		//Success
		IF NOT FB_MBReadInputs_Read.bBusy AND NOT FB_MBReadInputs_Read.bError THEN
			bRead := FALSE;
			bError := FALSE;
		END_IF	
		
		bRead := WORD_TO_BOOL(wRead);
	
	3: //Read Holding reg
		
		FB_MBReadRegs_Read(
		sIPAddr:= sIPAddr, 
		nTCPPort:= nTCPPort, 
		nUnitID:= nUnitID, 
		nQuantity:= 1 + nAddQuantity, 
		nMBAddr:= mBusAdr, 
		cbLength:= SIZEOF(aWordArrayRead), 
		pDestAddr:= ADR(aWordArrayRead), 
		bExecute:= bRead, 
		tTimeout:= tTimeout, 
		bBusy=> , 
		bError=> , 
		nErrId=> , 
		cbRead=> );
	
		//Error 
		IF FB_MBReadRegs_Read.bError THEN
			bRead := FALSE;
			bError := TRUE;
		END_IF
		
		//Success
		IF NOT FB_MBReadRegs_Read.bBusy AND NOT FB_MBReadRegs_Read.bError THEN
			bRead := FALSE;
			bError := FALSE;
		END_IF	
				
		//Skriv värdet
		IF bRead32bit THEN 
			IF bSwap THEN
				rRead := fWordToReal(aWordArrayRead);
			ELSE
				aWordArrayNoSwap[0] := aWordArrayRead[1];
				aWordArrayNoSwap[1] := aWordArrayRead[0];
 				rRead := fWordToReal(aWordArrayNoSwap);
			END_IF
		ELSE
			rRead := fSignedConverter(aWordArrayRead[0]);
		END_IF;
		
	4: //Read input registers
		
		FB_MBReadInputRegs_Read(
		sIPAddr:= sIPAddr, 
		nTCPPort:= nTCPPort, 
		nUnitID:= nUnitID, 
		nQuantity:= 1 + nAddQuantity, 
		nMBAddr:= mBusAdr, 
		cbLength:= SIZEOF(aWordArrayRead), 
		pDestAddr:= ADR(aWordArrayRead), 
		bExecute:= bRead, 
		tTimeout:= tTimeout, 
		bBusy=> , 
		bError=> , 
		nErrId=> , 
		cbRead=> );
	
		//Error 
		IF FB_MBReadInputRegs_Read.bError THEN
			bRead := FALSE;
			bError := TRUE;
		END_IF
		
		//Success
		IF NOT FB_MBReadInputRegs_Read.bBusy AND NOT FB_MBReadInputRegs_Read.bError THEN
			bRead := FALSE;
			bError := FALSE;
		END_IF	
	
		//Skriv värdet
		IF bRead32bit THEN 
			IF bSwap THEN
				rRead := fWordToReal(aWordArrayRead);
			ELSE
				aWordArrayNoSwap[0] := aWordArrayRead[1];
				aWordArrayNoSwap[1] := aWordArrayRead[0];
 				rRead := fWordToReal(aWordArrayNoSwap);
			END_IF
		ELSE
			rRead := fSignedConverter(aWordArrayRead[0]);
		END_IF;

END_CASE

bBusy := FB_MBReadCoils_Read.bBusy OR FB_MBReadInputs_Read.bBusy OR FB_MBReadRegs_Read.bBusy OR FB_MBReadInputRegs_Read.bBusy;

END_FUNCTION_BLOCK

// oaksModbusLibrary/Datahantering/fWordToReal
//OAKS AB
//2020-03-18
//Funtionsblock för att lägga ihop två separata word till en real 
FUNCTION fWordToReal : REAL
VAR_INPUT

wAwords : ARRAY  [0..1] OF WORD;
END_VAR
VAR
	union1 : uRealToTwoWORD;
END_VAR

union1.wTest[0] := wAwords[0];
union1.wTest[1] := wAwords[1];

fWordToReal := union1.rTest;

END_FUNCTION

// oaksModbusLibrary/Datahantering/fbReadWriteCoilRegBool
//Oaks AB
//2022-08-22
//Funktionsblock för läsning av coil register (modbus funktion 15). Värde skrivs endast då skriv värde avviker från återläst värde. Används ej på EEPROM minnen, då det riskerar att skriva sönder dem. Använd istället block med återläsning av värden.
//Läsning och skrivning sker i sekvens.
//Två larmutgångar. En via puls kopplas till tex. en TOF för egen larmhantering. En via inställd larmtid. Skall summalarm i skåp tändas vid fel kopplas någon av utgångarna till externt fbAlarm. 

FUNCTION_BLOCK fbReadWriteCoilRegBool
VAR_INPUT
	sIPAddr : STRING := ''; //Ip-adress
	nTCPPort : UINT; //Port
	nUnitID : UINT; //Modbus-ID
	mBusAdr : UINT; //Holding adress att läsa/skriva
	bEnable : BOOL := TRUE; //Flanktriggad
	tTimeout : TIME := T#5S;
	bBool : BOOL := FALSE; //Värde att skriva
			
END_VAR
VAR_OUTPUT
	bError : BOOL; //Puls (Använd för egen larmhantering)
	bBusy : BOOL; //Upptagen
	bSuccess : BOOL := FALSE; //Lyckad cykel
END_VAR

VAR
	bEnableInternal : BOOL := TRUE;
	iStep : INT := 0;
	fbReadRegs_1: FB_MBReadCoils;
	fbWriteCoils_Write: FB_MBWriteCoils;
	bRead : BOOL; //Värde återläst
	bWrite : BOOL; //Värde att skriva
	R_TRIG_Start : R_TRIG; 

	FB_MBWriteSingleCoil_Write: INT;
	
END_VAR

//Flanktriggning
R_TRIG_Start(CLK:= bEnable, Q=> bEnableInternal);

//Läs och skriv värden
CASE iStep OF
	
	0: //Start
		bSuccess := FALSE;
		bBusy := FALSE;
		
		IF bEnableInternal THEN
			iStep := 1;
			bError := FALSE;
		END_IF
		
	1: //Läs data
		bBusy := TRUE;
		
		fbReadRegs_1(
				sIPAddr:= sIPAddr, 
				nTCPPort:= INT_TO_UINT(nTCPPort), 
				nUnitID:= INT_TO_BYTE(nUnitID), 
				nQuantity:= 1, 
				nMBAddr:= UINT_TO_WORD(mBusAdr), 
				cbLength:= SIZEOF(bRead), 
				pDestAddr:= ADR(bRead), 
				bExecute:= TRUE,
				tTimeout:= tTimeout, 
				bBusy=> , 
				bError=> , 
				nErrId=> , 
				cbRead=> );
				
		//Error 
		IF fbReadRegs_1.bError THEN
			fbReadRegs_1(bExecute := FALSE);
			iStep := 99;
		END_IF
	
		//Gå till nästa steg
		IF NOT fbReadRegs_1.bBusy AND NOT fbReadRegs_1.bError THEN
			fbReadRegs_1(bExecute := FALSE);
			bError := FALSE;
			iStep := 2;
		END_IF;

	2: //Skriv data
	
		bWrite := bBool;
	
			//15 Force Multiple Coils
			IF bWrite <> bRead THEN
				fbWriteCoils_Write.bExecute := TRUE;
			ELSE
				fbWriteCoils_Write.bExecute := FALSE;
			END_IF;
			
				fbWriteCoils_Write(
					sIPAddr:= sIPAddr, 
					nTCPPort:= INT_TO_UINT(nTCPPort), 
					nUnitID:= INT_TO_BYTE(nUnitID), 
					nQuantity:= 1, 
					nMBAddr:= UINT_TO_WORD(mBusAdr),
					cbLength:= SIZEOF(bWrite), 
					pSrcAddr:= ADR(bWrite), 
					bExecute:= , 
					tTimeout:= tTimeout, 
					bBusy=> , 
					bError=> , 
					nErrId=> );
			
			//Felhantering
			IF fbWriteCoils_Write.bError THEN
				fbWriteCoils_Write(bExecute := FALSE);
				iStep := 99;
			END_IF
			
			//Nästa steg
			IF NOT fbWriteCoils_Write.bBusy AND NOT fbWriteCoils_Write.bError THEN
				fbWriteCoils_Write(bExecute := FALSE);
				bError := FALSE;
				bSuccess := TRUE; //Lyckad cykel
				iStep := 0;
			END_IF;
				
		99: //Felhantering total
			bError := TRUE;
			iStep := 0;
END_CASE

END_FUNCTION_BLOCK

// oaksModbusLibrary/Datahantering/fbReadWriteHoldingRegReal
//Oaks AB
//2022-02-08
//Funktionsblock för läsning av holding register. Värde skrivs endast då skriv värde avviker från återläst värde. Används ej på EEPROM minnen, då det riskerar att skriva sönder dem. Använd istället block med återläsning av värden.
//Real med skalning direkt anges på block, med inbyggd hantering av negativa värden. Läsning och skrivning sker i sekvens.
//Två larmutgångar. En via puls kopplas till tex. en TOF för egen larmhantering. En via inställd larmtid. Skall summalarm i skåp tändas vid fel kopplas någon av utgångarna till externt fbAlarm. 

FUNCTION_BLOCK fbReadWriteHoldingRegReal
VAR_INPUT
	sIPAddr : STRING := ''; //Ip-adress
	nTCPPort : UINT; //Port
	nUnitID : UINT; //Modbus-ID
	mBusAdr : UINT; //Holding adress att läsa/skriva
	bEnable : BOOL := TRUE; //Flanktriggad
	tTimeout : TIME := T#5S;
	rReal : REAL := 0; //Värde att skriva
	uiFaktor : REAL := 1; //Skalning
	
END_VAR
VAR_OUTPUT
	bError : BOOL; //Puls (Använd för egen larmhantering)
	bBusy : BOOL; //Upptagen
	bSuccess : BOOL := FALSE; //Lyckad cykel
END_VAR

VAR
	bEnableInternal : BOOL := TRUE;
	iStep : INT := 0;
	fbReadRegs_1: FB_MBReadRegs;
	fbWriteSingleReg_1: FB_MBWriteSingleReg;
	wRead : WORD; //Värde återläst
	wWrite : WORD; //Värde att skriva
	R_TRIG_Start : R_TRIG; 
END_VAR

//Flanktriggning
R_TRIG_Start(CLK:= bEnable, Q=> bEnableInternal);

//Läs och skriv värden
CASE iStep OF
	
	0: //Start
		bSuccess := FALSE;
		bBusy := FALSE;
		
		IF bEnableInternal THEN
			iStep := 1;
			bError := FALSE;
		END_IF
		
	1: //Läs data
		bBusy := TRUE;
		
		fbReadRegs_1(
				sIPAddr:= sIPAddr, 
				nTCPPort:= INT_TO_UINT(nTCPPort), 
				nUnitID:= INT_TO_BYTE(nUnitID), 
				nQuantity:= 1, 
				nMBAddr:= UINT_TO_WORD(mBusAdr), 
				cbLength:= SIZEOF(wRead), 
				pDestAddr:= ADR(wRead), 
				bExecute:= TRUE,
				tTimeout:= tTimeout, 
				bBusy=> , 
				bError=> , 
				nErrId=> , 
				cbRead=> );
	
		//Error 
		IF fbReadRegs_1.bError THEN
			fbReadRegs_1(bExecute := FALSE);
			iStep := 99;
		END_IF
	
		//Gå till nästa steg
		IF NOT fbReadRegs_1.bBusy AND NOT fbReadRegs_1.bError THEN
			fbReadRegs_1(bExecute := FALSE);
			bError := FALSE;
			iStep := 2;
		END_IF;

	2: //Skriv data
		//Konvertera REAL till WORD. 
		wWrite := fRealToWord(rReal, uiFaktor);
		//Skriv om värden skiljer sig
		IF wWrite <> wRead THEN
			fbWriteSingleReg_1(
				sIPAddr:= sIPAddr, 
				nTCPPort:= INT_TO_UINT(nTCPPort), 
				nUnitID:= INT_TO_BYTE(nUnitID), 
				nMBAddr:= UINT_TO_WORD(mBusAdr),
				nValue:= wWrite, 
				bExecute:= TRUE, 
				tTimeout:= tTimeout , 
				bBusy=> , 
				bError=> , 
				nErrId=> );
		//Annars börja om
		ELSE 
			iStep := 0;
		END_IF;
		
		//Felhantering
		IF fbWriteSingleReg_1.bError THEN
			fbWriteSingleReg_1(bExecute := FALSE);
			iStep := 99;
		END_IF
		
		//Nästa steg
		IF NOT fbWriteSingleReg_1.bBusy AND NOT fbWriteSingleReg_1.bError THEN
			fbWriteSingleReg_1(bExecute := FALSE);
			bError := FALSE;
			bSuccess := TRUE; //Lyckad cykel
			iStep := 0;
		END_IF;
			
		99: //Felhantering total
			bError := TRUE;
			iStep := 0;
END_CASE

END_FUNCTION_BLOCK

// oaksModbusLibrary/EBM Papst/fbEbmPapst
//OAKS AB
//2023-06-28
//Ver. 1.0
//Modbusblock för ebmpapst fläkt.
FUNCTION_BLOCK fbEbmPapst
VAR_INPUT
	sIPAddr : STRING := ''; 
	nTCPPort : UINT;
	nUnitID : UINT :=1;
	iModbusLoop : INT :=1; //Modbusslinga
			
END_VAR
VAR_OUTPUT
	RPM AT %M* : REAL;//Varvtal~wp:[unit]RPM[format]0[trendoptions]i:300
	U1 AT %M* : REAL;//Spänning~wp:[unit]V[format]0[trendoptions]i:300
	I1 AT %M* : REAL;//Ampere~wp:[unit]A[format]0.0[trendoptions]i:300	
	P1 AT %M* : REAL;//Effekt~wp:[unit]kW[format]0.0[trendoptions]i:300		
	PV8 AT %M* : STRING;//Modbus konfiguering~wp:
	FAULT AT %M* : BOOL;//Kommunikationsfel~wp:[alarmoptions]p:2
	
END_VAR
VAR
	offset : UINT;
	rTemp1 : REAL;
	rTemp2 : REAL;
	bSekvensFlagga : BOOL;
			
	FB_MBReadRegs_ArrReadRegs1 : FB_MBReadRegs;
	FB_MBReadRegs_ArrReadRegs2 : FB_MBReadRegs;
	FB_MBReadRegs_ArrReadInputsRegs1 : FB_MBReadInputRegs;
	FB_MBReadRegs_ArrReadInputsRegs2 : FB_MBReadInputRegs;

	wArrReadRegs1 : ARRAY [0..0] OF WORD; //ReadRegs
	wArrReadRegs2 : ARRAY [0..1] OF WORD; //ReadRegs
	wArrReadInputsRegs1 : ARRAY [0..9] OF WORD; //ReadInputsRegs
	wArrReadInputsRegs2 : ARRAY [0..9] OF WORD; //ReadInputsRegs
		
	//Kommunikationsfel
	fbKommTof : tof; 
	fbKommTon : fbAlarm;
	
	sIP: STRING(255);
	sPort: STRING(255);
	sModbusID: STRING(255);
	sModbusLoop: STRING(255);
	sTemp : STRING(255);
	
END_VAR

//General
	offset := 0;
//Sekvens	
	bSekvensFlagga := oaksGVL.aBModbusSekvens[iModbusLoop] = UINT_TO_INT(nUnitID);
//Modbus konfiguering
	sIP := CONCAT (SIPAddr, '');
	sPort := CONCAT ('<br>Port: ', UINT_TO_STRING(nTCPPort)); 								
	sModbusID := CONCAT('<br>ID: ', UINT_TO_STRING(nUnitID));
	sModbusLoop := CONCAT('<br>Loop: ', INT_TO_STRING(iModbusLoop));	

	sTemp := sIP;
	sTemp := CONCAT(sTemp, sPort);
	sTemp := CONCAT(sTemp, sModbusID);
	sTemp := CONCAT(sTemp, sModbusLoop);
	
	PV8 := sTemp;

///////////////		
//READ
///////////////		
	
	//Read Register D119
	FB_MBReadRegs_ArrReadRegs1(
	sIPAddr:= sIpAddr, 
	nTCPPort:= (nTCPPort),
	nUnitID:= UINT_TO_BYTE(nUnitID),  
	nQuantity:= 1, 
	nMBAddr:= 53529 + offset, 
	cbLength:= SIZEOF(wArrReadRegs1),  
	pDestAddr:= ADR(wArrReadRegs1), 
	bExecute:= bSekvensFlagga, 
	tTimeout:= T#10S, 
	bBusy=> , 
	bError=> , 
	nErrId=> , 
	cbRead=> );

	//Read Register D1A0-D1A1
	FB_MBReadRegs_ArrReadRegs2(
	sIPAddr:= sIpAddr, 
	nTCPPort:= (nTCPPort),
	nUnitID:= UINT_TO_BYTE(nUnitID),  
	nQuantity:= 2, 
	nMBAddr:= 53664 + offset, 
	cbLength:= SIZEOF(wArrReadRegs2),  
	pDestAddr:= ADR(wArrReadRegs2), 
	bExecute:= bSekvensFlagga, 
	tTimeout:= T#10S, 
	bBusy=> , 
	bError=> , 
	nErrId=> , 
	cbRead=> );	

	//Read Inputs D010-D019
	FB_MBReadRegs_ArrReadInputsRegs1(
	sIPAddr:= sIpAddr, 
	nTCPPort:= (nTCPPort), 
	nUnitID:= UINT_TO_BYTE(nUnitID), 
	nQuantity:= 9, 
	nMBAddr:= 53264 + offset,
	cbLength:= SIZEOF(wArrReadInputsRegs1), 
	pDestAddr:= ADR(wArrReadInputsRegs1), 
	bExecute:= bSekvensFlagga,
	tTimeout:= T#10S, 
	bBusy=> , 
	bError=> , 
	nErrId=> , 
	cbRead=> );	
	
	//Read Inputs D01A-D023
	FB_MBReadRegs_ArrReadInputsRegs2(
	sIPAddr:= sIpAddr, 
	nTCPPort:= (nTCPPort), 
	nUnitID:= UINT_TO_BYTE(nUnitID), 
	nQuantity:= 9, 
	nMBAddr:= 53274 + offset,
	cbLength:= SIZEOF(wArrReadInputsRegs2), 
	pDestAddr:= ADR(wArrReadInputsRegs2), 
	bExecute:= bSekvensFlagga,
	tTimeout:= T#10S, 
	bBusy=> , 
	bError=> , 
	nErrId=> , 
	cbRead=> );		

		//Values
		RPM := ((wArrReadInputsRegs1[0]*wArrReadRegs1[0])/64000); //D010 - Actual speed, Res.:1, Unit:rpm
		//wArrReadInputsRegs1[1]; //D011 - Notor status, Res.:-, Unit:-
		//wArrReadInputsRegs1[2]; //D012 - Warning, Res.:-, Unit:-
		U1 := (((wArrReadInputsRegs1[3]*(wArrReadRegs2[0]*20))/256)*0.001); //D013 - DC-link voltage, Res.:1, Unit:V
		I1 := (((wArrReadInputsRegs1[4]*(wArrReadRegs2[1]*2))/256)*0.001); //D014 - DC-link current, Res.:0.1, Unit:A
		//wArrReadInputsRegs1[5]; //D015 - Modul temperature, Res.:0.1, Unit:ºC
		//wArrReadInputsRegs1[6]; //D016 - Motor temperature, Res.:0.1, Unit:ºC
		//wArrReadInputsRegs1[7]; //D017 - Electronics temperature, Res.:0.1, Unit:ºC
		//wArrReadInputsRegs1[8]; //D018 - Current direction of rotation, Res.:-, Unit:-
		//wArrReadInputsRegs1[9]; //D019 - Current modulation level, Res.:-, Unit:-
	
		//wArrReadInputsRegs2[0]; //D01A - Current set value, Res.:-, Unit:-
		//wArrReadInputsRegs2[1]; //D01B - Actual sensor value, Res.:-, Unit:-
		//wArrReadInputsRegs2[2]; //D01C - Enable input status, Res.:-, Unit:-
		//wArrReadInputsRegs2[3]; //D01D - Current parameter set, Res.:-, Unit:-
		//wArrReadInputsRegs2[4]; //D01E - Current contol function, Res.:-, Unit:-
		//wArrReadInputsRegs2[5]; //D01F - Reserved, Res.:-, Unit:-
		//wArrReadInputsRegs2[6]; //D020 - Reserved, Res.:-, Unit:-
		rTemp1 := ((wArrReadRegs2[0]*20)*0.001);
		rTemp2 := ((wArrReadRegs2[1]*2)*0.001);
		P1 := ((((wArrReadInputsRegs2[7]*rTemp1)*rTemp2)/65536)*0.001); //D021 - Current power, Res.:0.1, Unit:kW 
		//wArrReadInputsRegs2[8]; //D022 - Reserved, Res.:-, Unit:-
		//wArrReadInputsRegs2[9]; //D023 - Acyual sensor value 1, Res.:-, Unit:-
	
//Communication error
	fbKommTof(IN:=FB_MBReadRegs_ArrReadInputsRegs1.bError , PT:=T#60S , Q=> , ET=> );
	fbKommTon(bInput:=fbKommTof.Q , tAlarmDelay:=T#20M , bAutoReset:= , bAlarmOutput=> );
	FAULT :=fbKommTon.bAlarmOutput;
		
//Write busy	
	oaksgvl.aBModbusBusyFlagga[iModbusLoop,nUnitID] := FB_MBReadRegs_ArrReadInputsRegs1.bBusy;

END_FUNCTION_BLOCK

// oaksModbusLibrary/EcoGuard/fbEcocomTemperature
//OAKS AB
//2020-03-18
// Funktionsblock för kommunikation  rumstemperatur från Ecoguard Ecocom
FUNCTION_BLOCK fbEcocomTemperature
VAR_INPUT
	sIpNUmber									: STRING(32);						// Ip nummer för Slav
	nTcpPort									: UINT := 502;					// Modbus port
	nUnitID 									: BYTE := 1;
	nAdressMaxTemperature						: UINT; 
	nAdressAvgTemperature						: UINT; 
	nAdressMinTemperature						: UINT; 
	tCommAlarmDelay : TIME := T#30M; // Tid för kommunikationsfelslarm.
	tToggleTime 	: TIME := T#60S; // ange hur ofta frågor skall ställas till Elvacon.
	tTimeout 		: TIME := T#58S; // inställd timeout-tid.
END_VAR
VAR_OUTPUT
	PV AT %M* : REAL;//Medel rumstemperatur hämtat från Ecoguard Ecocom~wp:[unit]°C[format]0.0[trendoptions]i:300
	PV1 AT %M* : REAL;//Högsta rumstemperatur hämtat från Ecoguard Ecocom~wp:[unit]°C[format]0.0[trendoptions]i:300
	PV2 AT %M* : REAL;//Lägsta rumstemperatur hämtat från Ecoguard Ecocom~wp:[unit]°C[format]0.0[trendoptions]i:300
	FAULT AT %M* : BOOL;//Kommunikationsfel~wp:
	PV8 AT %M* : STRING;//Modbus konfiguering~wp:
END_VAR
VAR
	rTemp : REAL;	

	sIP: STRING(255);
	sPort: STRING(255);
	sModbusID: STRING(255);
	sMaxtemp: STRING(255);
	sMedeltemp: STRING(255);
	sMintemp: STRING(255);
	sTemp : STRING(255);	

	fbKommTof : TOF;	
	fbKommTon : TON;
	FB_MBReadRegsAvg : FB_MBReadRegs;
	FB_MBReadRegsMax : FB_MBReadRegs;
	FB_MBReadRegsMin : FB_MBReadRegs;
	
	wInternalTempAvg : 	WORD; 
	wInternalTempMax : 	WORD; 
	wInternalTempMin : 	WORD; 
	fbToggle01: fbToggle;
	
END_VAR

//Modbus konfiguering
	sIP := CONCAT (sIpNUmber, '');
	sPort := CONCAT ('<br>Port: ', UINT_TO_STRING(nTCPPort)); 	
	sMaxtemp := CONCAT('<br>Adress maxtemperatur: ', INT_TO_STRING(nAdressMaxTemperature));						
	sMedeltemp := CONCAT('<br>Adress medeltemperatur: ', INT_TO_STRING(nAdressAvgTemperature));	
	sMintemp := CONCAT('<br>Adress mintemperatur: ', INT_TO_STRING(nAdressMinTemperature));
	
	sTemp := sIP;
	sTemp := CONCAT(sTemp, sPort);
	sTemp := CONCAT(sTemp, sMaxtemp);
	sTemp := CONCAT(sTemp, sMedeltemp);
	sTemp := CONCAT(sTemp, sMintemp);
	
	PV8 := sTemp;

	fbToggle01(bStart:=TRUE , tTimeOn:=tToggleTime , tTimeOff:=tToggleTime , bOutput=> );

	fbKommTof(IN:=FB_MBReadRegsAvg.bError OR FB_MBReadRegsMin.bError OR FB_MBReadRegsMax.bError , PT:=T#20S , Q=> , ET=> );
	fbKommTon(IN:=fbKommTof.Q , PT:=tCommAlarmDelay , Q=>FAULT , ET=> );
	// Hämta medel temperatur
	FB_MBReadRegsAvg(
	sIPAddr:= sIpNUmber, 
	nTCPPort:=nTcpPort , 
	nUnitID:=nUnitID , 
	nQuantity:=1 , 
	nMBAddr:= nAdressAvgTemperature, 
	cbLength:=SIZEOF(wInternalTempAvg) , 
	pDestAddr:=ADR(wInternalTempAvg) , 
	bExecute:=fbToggle01.bOutput , 
	tTimeout:=tTimeout , 
	bBusy=> , 
	bError=> , 
	nErrId=> , 
	cbRead=> );
	
	rTemp := fSignedConverter(wInternalTempAvg); 
	
	PV := rTemp / 10;
	// Hämta max temperatur
	FB_MBReadRegsMax(
	sIPAddr:= sIpNUmber, 
	nTCPPort:=nTcpPort , 
	nUnitID:=nUnitID , 
	nQuantity:=1 , 
	nMBAddr:= nAdressMaxTemperature, 
	cbLength:=SIZEOF(wInternalTempMax) , 
	pDestAddr:=ADR(wInternalTempMax) , 
	bExecute:=fbToggle01.bOutput , 
	tTimeout:=tTimeout , 
	bBusy=> , 
	bError=> , 
	nErrId=> , 
	cbRead=> );
	
	rTemp := fSignedConverter(wInternalTempMax); 
	
	PV1 := rTemp / 10;
	
	// Hämta min temperatur
	FB_MBReadRegsMin(
	sIPAddr:= sIpNUmber, 
	nTCPPort:=nTcpPort , 
	nUnitID:=nUnitID , 
	nQuantity:=1 , 
	nMBAddr:= nAdressMinTemperature, 
	cbLength:=SIZEOF(wInternalTempMin) , 
	pDestAddr:=ADR(wInternalTempMin) , 
	bExecute:=fbToggle01.bOutput , 
	tTimeout:=tTimeout , 
	bBusy=> , 
	bError=> , 
	nErrId=> , 
	cbRead=> );
	
	rTemp := fSignedConverter(wInternalTempMin); 
	
	PV2 := rTemp / 10;

END_FUNCTION_BLOCK

// oaksModbusLibrary/Elvaco/CME3100/Givare/fbElvacoTemperature
//OAKS AB
//2020-03-18
// Funktionsblock för kommunikation  via four-byte swapped float rumstemperatur från Elvaco CME3100
FUNCTION_BLOCK fbElvacoTemperature
VAR_INPUT
	sIpNUmber								: 		STRING(32);						// Ip nummer för Slav
	nTcpPort								: 		UINT := 502;					// Modbus port
	iModbusLoop : REFERENCE TO INT := 0; // Vill man att läsningarna ska ske givare för givare skapa en INT-variabel med värdet 16 som du sedan knyter hit. Läsningarna kommer då att ske efter modbussekvens 16. Knyter man inget här läses värdena efter inställd tid i tToggleTime samtidigt vilket kan bli problematiskt vid väldigt många samtidiga läsningar.
	nAdressTemperature						: UINT; 
	tCommAlarmDelay : TIME := T#30M; // Tid för kommunikationsfelslarm.
	tToggleTime : TIME := T#60S; // ange hur ofta frågor skall ställas till Elvacon. Denna används inte om något är knutet till iModbusLoop.
	tTimeout : TIME := T#58S; // inställd timeout-tid. Knyter man något på iModbusLoop är timeout-tiden 5 sekunder innan den går vidare.
	iSecId : DINT := 0;//Sekundär-ID
END_VAR
VAR_OUTPUT
	PV AT %M* : REAL;//Rumstemperatur~wp:[unit]°C[format]0.0[trendoptions]i:300
	FAULT AT %M* : BOOL;//Kommunikationsfel~wp:
	PV8 AT %M* : STRING;//Modbus konfiguering~wp:
END_VAR
VAR
	fbDifferenceCheckTemp: fbDifferenceCheck;
	fbAlarmTemp : fbAlarm;
	fbTonDifferenceCheck : TON;

	tTimeoutIntern : TIME;
	bStartaLasningTemperatur	: BOOL;

	bSekvensFlagga : BOOL;	

	sIP: STRING(255);
	sPort: STRING(255);
	sModbusID: STRING(255);
	sModbusLoop: STRING(255);
	sSecId : STRING(255);
	sTemp : STRING(255);

	fbKommTof : TOF;	
	fbKommTon : TON;
	FB_MBReadRegs01 : FB_MBReadRegs;
	wInternalTemp : ARRAY[0..1] OF	WORD; 
	fbToggle01: fbToggle;
	
	uRealToTwoWORD01 : uRealToTwoWORD;
END_VAR
VAR PERSISTENT
	tAlarmDelayDifferenceCheck : TIME := T#48H;
END_VAR

VAR_INPUT PERSISTENT
	AREAT AT %M* : INT; //Yta rumstemperatur~wp:
END_VAR


	IF __ISVALIDREF(iModbusLoop) THEN 
		IF iModbusLoop < 16 OR iModbusLoop > 16 THEN
			iModbusLoop := 16;
		END_IF;
		bSekvensFlagga := oaksGVL.aBModbusSekvens[iModbusLoop] = UINT_TO_INT(nAdressTemperature);
		fbToggle01(bStart:=FALSE , tTimeOn:=tToggleTime , tTimeOff:=tToggleTime , bOutput=> );
		tTimeoutIntern := T#5S;
	ELSE
		fbToggle01(bStart:=TRUE , tTimeOn:=tToggleTime , tTimeOff:=tToggleTime , bOutput=> );
		tTimeoutIntern := tTimeout;
	END_IF;
	bStartaLasningTemperatur := bSekvensFlagga OR fbToggle01.bOutput;

//Modbus konfiguering
	sIP := CONCAT (sIpNUmber, '');
	sPort := CONCAT ('<br>Port: ', UINT_TO_STRING(nTCPPort)); 						
	sModbusLoop := CONCAT('<br>Adress: ', INT_TO_STRING(nAdressTemperature));
	sSecId := CONCAT('<br>Sekundär-Id: ', DINT_TO_STRING(iSecId));

	sTemp := sIP;
	sTemp := CONCAT(sTemp, sPort);
	sTemp := CONCAT(sTemp, sModbusLoop);
	
	//Sekundär-Id
	IF iSecID > 0 THEN
		sTemp := CONCAT(Stemp,sSecId);
	ELSE 
		sTemp := STemp;
	END_IF
		
	PV8 := sTemp;

	fbKommTof(IN:=FB_MBReadRegs01.bError , PT:=T#20S , Q=> , ET=> );
	fbKommTon(IN:=fbKommTof.Q , PT:=tCommAlarmDelay , Q=>FAULT , ET=> );
	
	fbDifferenceCheckTemp(rPv:=PV );
	fbTonDifferenceCheck(IN:=NOT fbDifferenceCheckTemp.bDifference , PT:=tAlarmDelayDifferenceCheck , Q=> , ET=> );
	fbAlarmTemp(bInput:= fbTonDifferenceCheck.Q OR fbKommTon.Q , tAlarmDelay:=T#0S , bAutoReset:=TRUE , bAlarmOutput=>FAULT);

	FB_MBReadRegs01(
	sIPAddr:= sIpNUmber, 
	nTCPPort:=nTcpPort , 
	nUnitID:=1 , 
	nQuantity:=2 , 
	nMBAddr:= nAdressTemperature, 
	cbLength:=SIZEOF(wInternalTemp) , 
	pDestAddr:=ADR(wInternalTemp) , 
	bExecute:=bStartaLasningTemperatur , 
	tTimeout:=tTimeoutIntern , 
	bBusy=> , 
	bError=> , 
	nErrId=> , 
	cbRead=> );
	
	uRealToTwoWORD01.wTest[0] :=wInternalTemp [0];
	uRealToTwoWORD01.wTest[1] :=wInternalTemp [1];
	PV := uRealToTwoWORD01.rTest;
	
IF __ISVALIDREF(iModbusLoop) THEN 
	//Write busy
	oaksgvl.aBModbusBusyFlaggaAdresser[iModbusLoop-15,nAdressTemperature] := FB_MBReadRegs01.bBusy;
END_IF

END_FUNCTION_BLOCK

// oaksModbusLibrary/Elvaco/CME3100/Givare/fbElvacoTemperatureCo2
FUNCTION_BLOCK fbElvacoTemperatureCo2 EXTENDS fbElvacoTemperature
VAR_INPUT
	nAdressCo2		: UINT; 
END_VAR
VAR_OUTPUT
	PV1 AT %M* : REAL;//Koldioxidhalt~wp:[unit]ppm[format]0[trendoptions]i:300
END_VAR
VAR
	FB_MBReadRegs02 : FB_MBReadRegs;
	
	wInternalCo2	 : ARRAY[0..1] OF	WORD; 
	uRealToTwoWORD02 : uRealToTwoWORD;
END_VAR

VAR_INPUT PERSISTENT
	AREACO2 AT %M* : INT; //Yta koldioxid~wp:
END_VAR

	SUPER^();

	FB_MBReadRegs02(
	sIPAddr:= sIpNUmber, 
	nTCPPort:=nTcpPort , 
	nUnitID:=1 , 
	nQuantity:=2 , 
	nMBAddr:= nAdressCo2, 
	cbLength:=SIZEOF(wInternalCo2) , 
	pDestAddr:=ADR(wInternalCo2) , 
	bExecute:=bStartaLasningTemperatur , 
	tTimeout:=tTimeoutIntern , 
	bBusy=> , 
	bError=> , 
	nErrId=> , 
	cbRead=> );
	
	uRealToTwoWORD02.wTest[0] :=wInternalCo2 [0];
	uRealToTwoWORD02.wTest[1] :=wInternalCo2 [1];
	PV1 := uRealToTwoWORD02.rTest;

END_FUNCTION_BLOCK

// oaksModbusLibrary/Elvaco/CME3100/Givare/fbElvacoTemperatureHumidity
FUNCTION_BLOCK fbElvacoTemperatureHumidity EXTENDS fbElvacoTemperature
VAR_INPUT
	nAdressHumidity		: UINT; 
END_VAR
VAR_OUTPUT
	PV1 AT %M* : REAL;//Fukthalt~wp:[unit]rH%[trendoptions]i:300
END_VAR
VAR
	FB_MBReadRegs02 : FB_MBReadRegs;
	
	wInternalHumidity	 : ARRAY[0..1] OF	WORD; 
	uRealToTwoWORD02 : uRealToTwoWORD;
END_VAR

VAR_INPUT PERSISTENT
	AREAH AT %M* : INT; //Yta fuktighet~wp:
END_VAR

	SUPER^();

	FB_MBReadRegs02(
	sIPAddr:= sIpNUmber, 
	nTCPPort:=nTcpPort , 
	nUnitID:=1 , 
	nQuantity:=2 , 
	nMBAddr:= nAdressHumidity, 
	cbLength:=SIZEOF(wInternalHumidity) , 
	pDestAddr:=ADR(wInternalHumidity) , 
	bExecute:=bStartaLasningTemperatur , 
	tTimeout:=tTimeoutIntern , 
	bBusy=> , 
	bError=> , 
	nErrId=> , 
	cbRead=> );
	
	uRealToTwoWORD02.wTest[0] :=wInternalHumidity [0];
	uRealToTwoWORD02.wTest[1] :=wInternalHumidity [1];
	PV1 := uRealToTwoWORD02.rTest;

END_FUNCTION_BLOCK

// oaksModbusLibrary/Elvaco/CME3100/Mätare/fbElvacoElectricMeter
//OAKS AB
//2020-05-12
//Funktionsblock för att läsa elmätare från Elvaco
FUNCTION_BLOCK fbElvacoElectricMeter
VAR_INPUT
	sIPAddr : STRING := ''; 
	nTCPPort : UINT;
	nAdressEnergy	: UINT;
	nAdressPower	: UINT; 
	tCommAlarmDelay : TIME := T#30M; // Tid för kommunikationsfelslarm.
	tToggleTime : TIME := T#10S; // ange hur ofta frågor skall ställas till Elvacon.
	tTimeout : TIME := T#8S; // inställd timeout-tid.
	iSecId : DINT := 0;//Sekundär-ID
	rScalePower : REAL :=1; //Skalning effekt
 	bActivateDifferenceCheck : BOOL := TRUE; // När denna är true utgår kommunikationsfelslarm ifall värdet ej ändrats på T#49D17H2M47S295MS (inställbart)
END_VAR
VAR_OUTPUT
	PV8 AT %M* : STRING;//Modbus konfiguering~wp:
	FAULT AT %M* : BOOL;//Kommunikationsfel~wp:
	PV AT %M* : REAL;//Energi~wp:[unit]kWh[format]0.0[trendoptions]i:300
	PV1 AT %M* : REAL;//Effekt~wp:[unit]kW[format]0.0[trendoptions]i:300
		
END_VAR
VAR
	fbDifferenceCheckValue: fbDifferenceCheck;
	fbAlarmValue : fbAlarm;	
	fbTonDifferenceCheck : TON;

	offset : WORD;
	rTemp : REAL;
	//iTemp : UINT;
	fbToggle01: fbToggle;	
	
	FB_MBReadRegs_Energy : FB_MBReadRegs;
	FB_MBReadRegs_Power : FB_MBReadRegs;
	
	rPowerRead : REAL;	
	
	//Kommunikationsfel
	fbKommTof : tof; 
	fbKommTon : fbAlarm;
	
	sIP: STRING(255);
	sPort: STRING(255);
	sModbusID: STRING(255);
	sModbusLoop: STRING(255);
	sTemp : STRING(255);
	sSecId : STRING(255);
END_VAR
VAR PERSISTENT
	tAlarmDelayDifferenceCheck : TIME := T#49D17H2M47S295MS;
END_VAR

//Modbus konfiguering
	sIP := CONCAT (sIPAddr, '');
	sPort := CONCAT ('<br>Port: ', UINT_TO_STRING(nTCPPort));
	sSecId := CONCAT('<br>Sekundär-Id: ', DINT_TO_STRING(iSecId));

	sTemp := sIP;
	sTemp := CONCAT(sTemp, sPort);
	sTemp := CONCAT(sTemp, sModbusLoop);
	
	//Sekundär-Id
	IF iSecID > 0 THEN
		sTemp := CONCAT(Stemp,sSecId);
	ELSE 
		sTemp := STemp;
	END_IF
		
	PV8 := sTemp;

///////////////		
//READ
///////////////		
	fbToggle01(bStart:=TRUE , tTimeOn:=tToggleTime , tTimeOff:=tToggleTime , bOutput=> );
	
	FB_MBReadRegs_Energy(
	sIPAddr:= sIpAddr, 
	nTCPPort:= INT_TO_UINT(nTCPPort), 
	nUnitID:= 1, 
	nQuantity:= 2, 
	nMBAddr:= nAdressEnergy + offset, 
	cbLength:= SIZEOF(PV), 
	pDestAddr:= ADR(PV), 
	bExecute:= fbToggle01.bOutput, 
	tTimeout:= tTimeout, 
	bBusy=> , 
	bError=> , 
	nErrId=> , 
	cbRead=> );
	
	FB_MBReadRegs_Power(
	sIPAddr:= sIpAddr, 
	nTCPPort:= INT_TO_UINT(nTCPPort), 
	nUnitID:= 1, 
	nQuantity:= 2, 
	nMBAddr:= nAdressPower + offset, 
	cbLength:= SIZEOF(rPowerRead), 
	pDestAddr:= ADR(rPowerRead), 
	bExecute:= fbToggle01.bOutput, 
	tTimeout:= tTimeout, 
	bBusy=> , 
	bError=> , 
	nErrId=> , 
	cbRead=> );
	
	//Skalning effekt då denna ofta kommer i W. 
	PV1 := rPowerRead * rScalePower;
	
//Communication error
	fbKommTof(IN:=FB_MBReadRegs_Energy.bError OR FB_MBReadRegs_Power.bError, PT:=T#20S , Q=> , ET=> );
	fbKommTon(bInput:=fbKommTof.Q , tAlarmDelay:=tCommAlarmDelay , bAutoReset:= , bAlarmOutput=> );
	fbDifferenceCheckValue(rPv:=PV );
	fbTonDifferenceCheck(IN:=NOT fbDifferenceCheckValue.bDifference , PT:=tAlarmDelayDifferenceCheck , Q=> , ET=> );
	fbAlarmValue(bInput:= (fbTonDifferenceCheck.Q AND bActivateDifferenceCheck) OR fbKommTon.bAlarmOutput, tAlarmDelay:=T#0S , bAutoReset:=TRUE , bAlarmOutput=>FAULT);

END_FUNCTION_BLOCK

// oaksModbusLibrary/Elvaco/CME3100/Mätare/fbElvacoElectricMeterEnergy
//OAKS AB
//2020-05-12
//Funktionsblock för att läsa elmätare från Elvaco
FUNCTION_BLOCK fbElvacoElectricMeterEnergy
VAR_INPUT
	sIPAddr : STRING := ''; 
	nTCPPort : UINT;
	nAdressEnergy	: UINT;
	tCommAlarmDelay : TIME := T#30M; // Tid för kommunikationsfelslarm.
	tToggleTime : TIME := T#10S; // ange hur ofta frågor skall ställas till Elvacon.
	tTimeout : TIME := T#8S; // inställd timeout-tid.
	iSecId : DINT := 0;//Sekundär-ID
	rScalePower : REAL :=1; //Skalning effekt
 	bActivateDifferenceCheck : BOOL := TRUE; // När denna är true utgår kommunikationsfelslarm ifall värdet ej ändrats på T#49D17H2M47S295MS (inställbart)
END_VAR
VAR_OUTPUT
	PV8 AT %M* : STRING;//Modbus konfiguering~wp:
	FAULT AT %M* : BOOL;//Kommunikationsfel~wp:
	PV AT %M* : REAL;//Energi~wp:[unit]kWh[format]0.0[trendoptions]i:300
			
END_VAR
VAR
	fbDifferenceCheckValue: fbDifferenceCheck;
	fbAlarmValue : fbAlarm;		
	fbTonDifferenceCheck : TON;
	offset : WORD;
	rTemp : REAL;
	//iTemp : UINT;
	fbToggle01: fbToggle;	
	
	FB_MBReadRegs_Energy : FB_MBReadRegs;
	
	//Kommunikationsfel
	fbKommTof : tof; 
	fbKommTon : fbAlarm;
	
	sIP: STRING(255);
	sPort: STRING(255);
	sModbusID: STRING(255);
	sModbusLoop: STRING(255);
	sTemp : STRING(255);
	sSecId : STRING(255);
END_VAR
VAR PERSISTENT
	tAlarmDelayDifferenceCheck : TIME := T#49D17H2M47S295MS;
END_VAR

//Modbus konfiguering
	sIP := CONCAT (sIPAddr, '');
	sPort := CONCAT ('<br>Port: ', UINT_TO_STRING(nTCPPort));
	sSecId := CONCAT('<br>Sekundär-Id: ', DINT_TO_STRING(iSecId));

	sTemp := sIP;
	sTemp := CONCAT(sTemp, sPort);
	sTemp := CONCAT(sTemp, sModbusLoop);
	
	//Sekundär-Id
	IF iSecID > 0 THEN
		sTemp := CONCAT(Stemp,sSecId);
	ELSE 
		sTemp := STemp;
	END_IF
		
	PV8 := sTemp;

///////////////		
//READ
///////////////		
	fbToggle01(bStart:=TRUE , tTimeOn:=tToggleTime , tTimeOff:=tToggleTime , bOutput=> );
	
	FB_MBReadRegs_Energy(
	sIPAddr:= sIpAddr, 
	nTCPPort:= INT_TO_UINT(nTCPPort), 
	nUnitID:= 1, 
	nQuantity:= 2, 
	nMBAddr:= nAdressEnergy + offset, 
	cbLength:= SIZEOF(PV), 
	pDestAddr:= ADR(PV), 
	bExecute:= fbToggle01.bOutput, 
	tTimeout:= tTimeout, 
	bBusy=> , 
	bError=> , 
	nErrId=> , 
	cbRead=> );
	
//Communication error
	fbKommTof(IN:=FB_MBReadRegs_Energy.bError, PT:=T#20S , Q=> , ET=> );
	fbKommTon(bInput:=fbKommTof.Q , tAlarmDelay:=tCommAlarmDelay , bAutoReset:= , bAlarmOutput=> );
	fbDifferenceCheckValue(rPv:=PV );
	fbTonDifferenceCheck(IN:=NOT fbDifferenceCheckValue.bDifference , PT:=tAlarmDelayDifferenceCheck , Q=> , ET=> );
	fbAlarmValue(bInput:= (fbTonDifferenceCheck.Q AND bActivateDifferenceCheck) OR fbKommTon.bAlarmOutput, tAlarmDelay:=T#0S , bAutoReset:=TRUE , bAlarmOutput=>FAULT);

END_FUNCTION_BLOCK

// oaksModbusLibrary/Elvaco/CME3100/Mätare/fbElvacoEnergyMeter
//OAKS AB
//2020-05-12
//Funktionsblock för att läsa energimätare från Elvaco
FUNCTION_BLOCK fbElvacoEnergyMeter
VAR_INPUT
	sIPAddr : STRING := ''; 
	nTCPPort : UINT;
	nAdressEnergy						: UINT; 
	nAdressPower						: UINT; 
	nAdressSuptemp						: UINT;	
	nAdressRettemp						: UINT;	
	tCommAlarmDelay : TIME := T#30M; // Tid för kommunikationsfelslarm.
	tToggleTime : TIME := T#10S; // ange hur ofta frågor skall ställas till Elvacon.
	tTimeout : TIME := T#8S; // inställd timeout-tid.
	iSecId : DINT := 0;//Sekundär-ID
	bActivateDifferenceCheck : BOOL := TRUE; // När denna är true utgår kommunikationsfelslarm ifall värdet ej ändrats på T#48H (inställbart)
END_VAR
VAR_OUTPUT
	PV8 AT %M* : STRING;//Modbus konfiguering~wp:
	FAULT AT %M* : BOOL;//Kommunikationsfel~wp:
	PV AT %M* : REAL;//Energi~wp:[unit]MWh[format]0.000[trendoptions]i:300
	PV1 AT %M* : REAL;//Effekt~wp:[unit]kW[format]0.0[trendoptions]i:300
	SUPTEMP_PV AT %M* : REAL;//Framledningstemperatur~wp:[unit]°C[format]0.0[trendoptions]i:300
	RETTEMP_PV AT %M* : REAL;//Returledningstemperatur~wp:[unit]°C[format]0.0[trendoptions]i:300
END_VAR
VAR
	fbDifferenceCheckValue: fbDifferenceCheck;
	fbAlarmValue : fbAlarm;	
	fbTonDifferenceCheck : TON;
	offset : WORD;
	rTemp : REAL;
	//iTemp : UINT;
	fbToggle01: fbToggle;	
	
	FB_MBReadRegs_Energy : FB_MBReadRegs;
	FB_MBReadRegs_Power : FB_MBReadRegs;
	FB_MBReadRegs_Suptemp: FB_MBReadRegs;
	FB_MBReadRegs_Rettemp: FB_MBReadRegs;
		
	//Kommunikationsfel
	fbKommTof : tof; 
	fbKommTon : fbAlarm;
	
	sIP: STRING(255);
	sPort: STRING(255);
	sModbusID: STRING(255);
	sModbusLoop: STRING(255);
	sTemp : STRING(255);
	sSecId : STRING(255);
END_VAR
VAR PERSISTENT
	tAlarmDelayDifferenceCheck : TIME := T#48H;
END_VAR

//Modbus konfiguering
	sIP := CONCAT (sIPAddr, '');
	sPort := CONCAT ('<br>Port: ', UINT_TO_STRING(nTCPPort));
	sSecId := CONCAT('<br>Sekundär-Id: ', DINT_TO_STRING(iSecId));

	sTemp := sIP;
	sTemp := CONCAT(sTemp, sPort);
	sTemp := CONCAT(sTemp, sModbusLoop);
	
	//Sekundär-Id
	IF iSecID > 0 THEN
		sTemp := CONCAT(Stemp,sSecId);
	ELSE 
		sTemp := STemp;
	END_IF
		
	PV8 := sTemp;

///////////////		
//READ
///////////////		
	fbToggle01(bStart:=TRUE , tTimeOn:=tToggleTime , tTimeOff:=tToggleTime , bOutput=> );
	
	FB_MBReadRegs_Energy(
	sIPAddr:= sIpAddr, 
	nTCPPort:= INT_TO_UINT(nTCPPort), 
	nUnitID:= 1, 
	nQuantity:= 2, 
	nMBAddr:= nAdressEnergy + offset, 
	cbLength:= SIZEOF(PV), 
	pDestAddr:= ADR(PV), 
	bExecute:= fbToggle01.bOutput, 
	tTimeout:= tTimeout, 
	bBusy=> , 
	bError=> , 
	nErrId=> , 
	cbRead=> );
	
	FB_MBReadRegs_Power(
	sIPAddr:= sIpAddr, 
	nTCPPort:= INT_TO_UINT(nTCPPort), 
	nUnitID:= 1, 
	nQuantity:= 2, 
	nMBAddr:= nAdressPower + offset, 
	cbLength:= SIZEOF(PV1), 
	pDestAddr:= ADR(PV1), 
	bExecute:= fbToggle01.bOutput, 
	tTimeout:= tTimeout, 
	bBusy=> , 
	bError=> , 
	nErrId=> , 
	cbRead=> );
	
	FB_MBReadRegs_Suptemp(
	sIPAddr:= sIpAddr, 
	nTCPPort:= INT_TO_UINT(nTCPPort), 
	nUnitID:= 1, 
	nQuantity:= 2, 
	nMBAddr:= nAdressSuptemp + offset, 
	cbLength:= SIZEOF(SUPTEMP_PV), 
	pDestAddr:= ADR(SUPTEMP_PV), 
	bExecute:= fbToggle01.bOutput, 
	tTimeout:= tTimeout, 
	bBusy=> , 
	bError=> , 
	nErrId=> , 
	cbRead=> );
	
	FB_MBReadRegs_Rettemp(
	sIPAddr:= sIpAddr, 
	nTCPPort:= INT_TO_UINT(nTCPPort), 
	nUnitID:= 1, 
	nQuantity:= 2, 
	nMBAddr:= nAdressRettemp + offset, 
	cbLength:= SIZEOF(RETTEMP_PV), 
	pDestAddr:= ADR(RETTEMP_PV), 
	bExecute:= fbToggle01.bOutput, 
	tTimeout:= tTimeout, 
	bBusy=> , 
	bError=> , 
	nErrId=> , 
	cbRead=> );
	
//Communication error
	fbKommTof(IN:=FB_MBReadRegs_Energy.bError , PT:=T#20S , Q=> , ET=> );
	fbKommTon(bInput:=fbKommTof.Q , tAlarmDelay:=tCommAlarmDelay , bAutoReset:= , bAlarmOutput=> );
	fbDifferenceCheckValue(rPv:=SUPTEMP_PV );
	fbTonDifferenceCheck(IN:=NOT fbDifferenceCheckValue.bDifference , PT:=tAlarmDelayDifferenceCheck , Q=> , ET=> );
	fbAlarmValue(bInput:= (fbTonDifferenceCheck.Q AND bActivateDifferenceCheck) OR fbKommTon.bAlarmOutput, tAlarmDelay:=T#0S , bAutoReset:=TRUE , bAlarmOutput=>FAULT);

END_FUNCTION_BLOCK

// oaksModbusLibrary/Elvaco/CME3100/Mätare/fbElvacoWaterMeter
//OAKS AB
//2020-05-12
//Funktionsblock för att läsa vattenmätare från Elvaco.
FUNCTION_BLOCK fbElvacoWaterMeter
VAR_INPUT
	sIPAddr : STRING := ''; 
	nTCPPort : UINT;
	nAdressVolume						: UINT; 
	tCommAlarmDelay : TIME := T#30M; // Tid för kommunikationsfelslarm.
	tToggleTime : TIME := T#10S; // ange hur ofta frågor skall ställas till Elvacon.
	tTimeout : TIME := T#8S; // inställd timeout-tid.
	iSecId : DINT := 0;//Sekundär-ID
	bActivateDifferenceCheck : BOOL := TRUE; // När denna är true utgår kommunikationsfelslarm ifall värdet ej ändrats på T#49D17H2M47S295MS (inställbart)
END_VAR
VAR_OUTPUT
	PV8 AT %M* : STRING;//Modbus konfiguering~wp:
	FAULT AT %M* : BOOL;//Kommunikationsfel~wp:
	PV AT %M* : REAL;//Volym~wp:[unit]m3[format]0.0[trendoptions]i:300
	
END_VAR
VAR
	fbDifferenceCheckValue: fbDifferenceCheck;
	fbAlarmValue : fbAlarm;			
	fbTonDifferenceCheck : TON;
	offset : WORD;
	rTemp : REAL;
	//iTemp : UINT;
	fbToggle01: fbToggle;	
	
	FB_MBReadRegs_Volume : FB_MBReadRegs;
			
	//Kommunikationsfel
	fbKommTof : tof; 
	fbKommTon : fbAlarm;
	
	sIP: STRING(255);
	sPort: STRING(255);
	sModbusID: STRING(255);
	sModbusLoop: STRING(255);
	sTemp : STRING(255);
	sSecId : STRING(255);
END_VAR
VAR PERSISTENT
	tAlarmDelayDifferenceCheck : TIME := T#49D17H2M47S295MS;
END_VAR

//Modbus konfiguering
	sIP := CONCAT (sIPAddr, '');
	sPort := CONCAT ('<br>Port: ', UINT_TO_STRING(nTCPPort));
	sSecId := CONCAT('<br>Sekundär-Id: ', DINT_TO_STRING(iSecId));

	sTemp := sIP;
	sTemp := CONCAT(sTemp, sPort);
	sTemp := CONCAT(sTemp, sModbusLoop);
	
	//Sekundär-Id
	IF iSecID > 0 THEN
		sTemp := CONCAT(Stemp,sSecId);
	ELSE 
		sTemp := STemp;
	END_IF
		
	PV8 := sTemp;

///////////////		
//READ
///////////////		
	fbToggle01(bStart:=TRUE , tTimeOn:=tToggleTime , tTimeOff:=tToggleTime , bOutput=> );
	
	FB_MBReadRegs_Volume(
	sIPAddr:= sIpAddr, 
	nTCPPort:= INT_TO_UINT(nTCPPort), 
	nUnitID:= 1, 
	nQuantity:= 2, 
	nMBAddr:= nAdressVolume + offset, 
	cbLength:= SIZEOF(PV), 
	pDestAddr:= ADR(PV), 
	bExecute:= fbToggle01.bOutput, 
	tTimeout:= tTimeout, 
	bBusy=> , 
	bError=> , 
	nErrId=> , 
	cbRead=> );
	
//Communication error
	fbKommTof(IN:=FB_MBReadRegs_Volume.bError , PT:=T#20S , Q=> , ET=> );
	fbKommTon(bInput:=fbKommTof.Q , tAlarmDelay:=tCommAlarmDelay , bAutoReset:= , bAlarmOutput=> );
	fbDifferenceCheckValue(rPv:=PV );
	fbTonDifferenceCheck(IN:=NOT fbDifferenceCheckValue.bDifference , PT:=tAlarmDelayDifferenceCheck , Q=> , ET=> );
	fbAlarmValue(bInput:= (fbTonDifferenceCheck.Q AND bActivateDifferenceCheck) OR fbKommTon.bAlarmOutput, tAlarmDelay:=T#0S , bAutoReset:=TRUE , bAlarmOutput=>FAULT);

END_FUNCTION_BLOCK

// oaksModbusLibrary/Elvaco/CME3100/fbElvacoGeneral
//OAKS AB
//2020-03-18
//Funktionsblock för läsning av four-byte swapped float från Elvaco CME3100
FUNCTION_BLOCK fbElvacoGeneral
VAR_INPUT
	sIPAddr : STRING := ''; 
	nTCPPort : UINT := 502;
	nUnitID : UINT := 1;
	nStartAdr : UINT := 1; //Startadress läsning
	rScale : REAL :=1; //Skalning (läst värde multipliceras med rScale)
	tCommAlarmDelay : TIME := T#30M; // Tid för kommunikationsfelslarm.
	tToggleTime : TIME := T#60S; // ange hur ofta frågor skall ställas till Elvacon.
	tTimeout : TIME := T#58S; // inställd timeout-tid.
	bActivateDifferenceCheck : BOOL := TRUE; // När denna är true utgår kommunikationsfelslarm ifall värdet ej ändrats på T#49D17H2M47S295MS (inställbart)
END_VAR
VAR_OUTPUT
	wRead : ARRAY [0..1] OF WORD;
	rPv : REAL; //Läst värde
	bAlarm : BOOL; //Kommunikationsfel
	bBusy : BOOL; //
	sModbusConfig AT %M* : STRING;//Modbus konfiguering sammanfattning ip-adress, tcp-port och adress i strängformat ~wp:
END_VAR
VAR
	fbDifferenceCheckValue: fbDifferenceCheck;
	fbAlarmValue : fbAlarm;	
	fbTonDifferenceCheck : TON;
	sIP: STRING(255);
	sPort: STRING(255);
	sModbusID: STRING(255);
	sModbusLoop: STRING(255);
	sTemp : STRING(255);	


	FB_MBReadRegs_1: FB_MBReadRegs;
	
	//Kommunikationsfel
	fbKommTof : tof; 
	fbKommTon : ton;
	
	fbToggle01: fbToggle;
END_VAR
VAR PERSISTENT
	tAlarmDelayDifferenceCheck : TIME := T#49D17H2M47S295MS;
END_VAR

//Modbus konfiguering
	sIP := CONCAT (sIPAddr, '');
	sPort := CONCAT ('<br>Port: ', UINT_TO_STRING(nTCPPort)); 						
	sModbusLoop := CONCAT('<br>Adress: ', INT_TO_STRING(nStartAdr));	

	sTemp := sIP;
	sTemp := CONCAT(sTemp, sPort);
	sTemp := CONCAT(sTemp, sModbusLoop);
	
	sModbusConfig := sTemp;

//Läs data

fbToggle01(bStart:=TRUE , tTimeOn:=tToggleTime , tTimeOff:=tToggleTime , bOutput=> );

FB_MBReadRegs_1(
	sIPAddr:= sIPAddr , 
	nTCPPort:= nTCPPort, 
	nUnitID:= UINT_TO_BYTE(nUnitID), 
	nQuantity:= 2, 
	nMBAddr:= nStartAdr, 
	cbLength:= SIZEOF(wRead), 
	pDestAddr:= ADR(wRead), 
	bExecute:= fbToggle01.bOutput , 
	tTimeout:= tTimeout, 
	bBusy=> , 
	bError=> , 
	nErrId=> , 
	cbRead=> );
	
	//Upptagen
	bBusy := FB_MBReadRegs_1.bBusy;
	
	//Konveterat läst värde
	rPv := fWordToReal(wRead) * rScale;
	
//Kommunikationsfel
	fbKommTof(IN:=FB_MBReadRegs_1.bError , PT:=T#20S , Q=> , ET=> );
	fbKommTon(IN:=fbKommTof.Q , PT:=tCommAlarmDelay, Q=> , ET=> );
	fbDifferenceCheckValue(rPv:=rPv );
	fbTonDifferenceCheck(IN:=NOT fbDifferenceCheckValue.bDifference , PT:=tAlarmDelayDifferenceCheck , Q=> , ET=> );
	fbAlarmValue(bInput:= (fbTonDifferenceCheck.Q AND bActivateDifferenceCheck) OR fbKommTon.Q, tAlarmDelay:=T#0S , bAutoReset:=TRUE , bAlarmOutput=>bAlarm);

END_FUNCTION_BLOCK

// oaksModbusLibrary/Eveco/fbEveco
//OAKS AB
//2020-05-12
//Block för fläktluftkylare Eveco med Modbus sabiana MB EXT EN Rev_10 modul
//Påbörjad färdigställs vid driftsättning
FUNCTION_BLOCK fbEveco
VAR_INPUT
	sIPAddr : STRING := ''; 
	nTCPPort : UINT;
	nUnitID : UINT :=1;
	iModbusLoop : INT :=1; //Modbusslinga
	bOnOffCommand : BOOL; // TRUE = ON FALSE = OFF
	usiSpeed : ANY; // Knyt variabel av typen USINT för att välja hastighet på fläkt (0-4). Lämnas input tom (dvs. ingenting knutet till den) så görs inga skrivningar utav detta.
END_VAR
VAR_OUTPUT
	OP AT %M* : REAL;//Styrsignal kyla~wp:[unit]%[format]0[trendoptions]i:300	
	V AT %M* : BOOL;//Driftindikering~wp:[trendoptions]i:14400, t:1
	PV8 AT %M* : STRING;//Modbus konfiguering~wp:
	FAULT AT %M* : BOOL;//Kommunikationsfel~wp:

	
	
	T3_PV AT %M* : REAL;//Temperatur värmebatteri~wp:[unit]°C[format]0.0[trendoptions]i:300	

	T1_PV AT %M* : REAL;//Rumstemperatur~wp:[unit]°C[format]0.0[trendoptions]i:300
	T1_HAL AT %M* : BOOL;//Hög rumstemperatur~wp:
	T1_LAL AT %M* : BOOL;//Låg rumstemperatur~wp:
	

END_VAR
VAR
	

	fbHightempAlarm : fbHighLimitAlarm;
	fbLowtempAlarm : fbLowLimitAlarm;

	offset : WORD;
	rTemp : REAL;
	iTemp : UINT;
	bSekvensFlagga : BOOL;
			
	FB_MBReadRegs_T1: FB_MBReadRegs;
	wT1 : WORD; //Holding
	
	FB_MBReadRegs_T3: FB_MBReadRegs;
	wT3: WORD; //Holding
	
	FB_MBReadRegs_MachineState: FB_MBReadRegs;
	wMachineState: WORD; //Holding
	
	FB_MBReadRegs_Op: FB_MBReadRegs;
	wOp: WORD; //Holding

	//Kommunikationsfel
	fbKommTof : tof; 
	fbKommTon : fbAlarm;
	
	sIP: STRING(255);
	sPort: STRING(255);
	sModbusID: STRING(255);
	sModbusLoop: STRING(255);
	sTemp : STRING(255);
	
	
	fbReadWriteHoldingReg_bStartStopp: fbReadWriteHoldingReg;
	fbReadWriteHoldingReg_usiSpeed : fbReadWriteHoldingReg;
	
	fbReadWriteHoldingRegSummerSetpoint: fbReadWriteHoldingReg;
	fbReadWriteHoldingRegWinterSetpoint: fbReadWriteHoldingReg;
	
	usiOutput : USINT;
END_VAR
VAR_INPUT PERSISTENT
	T1_SP  AT %M* : REAL := 19;//Börvärde~wp:[unit]°C[format]0.0
	T1_AHL AT %M* : REAL := 25;//Larmgräns hög temperatur~wp:[unit]°C[format]0.0
	T1_HAD AT %M* : REAL := 60;//Larmfördröjning hög temperatur~wp:[unit]min[format]0
	T1_ALL AT %M* : REAL := 15;//Larmgräns låg temperatur~wp:[unit]°C[format]0.0
	T1_LAD AT %M* : REAL := 60;//Larmfördröjning låg temperatur~wp:[unit]min[format]0
END_VAR

//General
	offset := 0;
//Sekvens	
	bSekvensFlagga := oaksGVL.aBModbusSekvens[iModbusLoop] = UINT_TO_INT(nUnitID);
//Modbus konfiguering
	sIP := CONCAT (SIPAddr, '');
	sPort := CONCAT ('<br>Port: ', UINT_TO_STRING(nTCPPort)); 								
	sModbusID := CONCAT('<br>ID: ', UINT_TO_STRING(nUnitID));
	sModbusLoop := CONCAT('<br>Loop: ', INT_TO_STRING(iModbusLoop));	

	sTemp := sIP;
	sTemp := CONCAT(sTemp, sPort);
	sTemp := CONCAT(sTemp, sModbusID);
	sTemp := CONCAT(sTemp, sModbusLoop);
	
	PV8 := sTemp;

///////////////		
//READ
///////////////		
	
	//Read Holding T1 temperatur
	FB_MBReadRegs_T1(
	sIPAddr:= sIpAddr, 
	nTCPPort:= INT_TO_UINT(nTCPPort), 
	nUnitID:= INT_TO_BYTE(nUnitID), 
	nQuantity:= 1, 
	nMBAddr:= 4098 + offset, 
	cbLength:= SIZEOF(wT1), 
	pDestAddr:= ADR(wT1), 
	bExecute:= bSekvensFlagga, 
	tTimeout:= T#3S, 
	bBusy=> , 
	bError=> , 
	nErrId=> , 
	cbRead=> );
	
	rTemp := WORD_TO_REAL(wT1);
	T1_PV := fSignedConverter(rTemp) / 10;
	
	//Read Holding T3 temperatur
	FB_MBReadRegs_T3(
	sIPAddr:= sIpAddr, 
	nTCPPort:= INT_TO_UINT(nTCPPort), 
	nUnitID:= INT_TO_BYTE(nUnitID), 
	nQuantity:= 1, 
	nMBAddr:= 4100 + offset, 
	cbLength:= SIZEOF(wT3), 
	pDestAddr:= ADR(wT3), 
	bExecute:= bSekvensFlagga, 
	tTimeout:= T#3S, 
	bBusy=> , 
	bError=> , 
	nErrId=> , 
	cbRead=> );
	
	rTemp := WORD_TO_REAL(wT3);
	T3_PV := fSignedConverter(rTemp) / 10;
	
	//Read Holding machine state
	FB_MBReadRegs_MachineState(
	sIPAddr:= sIpAddr, 
	nTCPPort:= INT_TO_UINT(nTCPPort), 
	nUnitID:= INT_TO_BYTE(nUnitID), 
	nQuantity:= 1, 
	nMBAddr:= 4111 + offset, 
	cbLength:= SIZEOF(wMachineState), 
	pDestAddr:= ADR(wMachineState), 
	bExecute:= bSekvensFlagga, 
	tTimeout:= T#3S, 
	bBusy=> , 
	bError=> , 
	nErrId=> , 
	cbRead=> );
	
	V := WORD_TO_BOOL(wMachineState);
	
	//Read Holding 0-10V  Analog output 0-10V
	FB_MBReadRegs_T3(
	sIPAddr:= sIpAddr, 
	nTCPPort:= INT_TO_UINT(nTCPPort), 
	nUnitID:= INT_TO_BYTE(nUnitID), 
	nQuantity:= 1, 
	nMBAddr:= 4134 + offset, 
	cbLength:= SIZEOF(wOp), 
	pDestAddr:= ADR(wOp), 
	bExecute:= bSekvensFlagga, 
	tTimeout:= T#3S, 
	bBusy=> , 
	bError=> , 
	nErrId=> , 
	cbRead=> );
	
	OP := WORD_TO_REAL(wOp);
	
(********************* Skrivningar *********************)
	fbReadWriteHoldingReg_bStartStopp(
	sIPAddr:= sIpAddr, 
	nTCPPort:= INT_TO_UINT(nTCPPort), 
	nUnitID:= INT_TO_BYTE(nUnitID), 
	mBusAdr:=4182 + offset, 
	bEnable:=bSekvensFlagga , 
	iWrite:= BOOL_TO_UINT(NOT bOnOffCommand), 
	iRead=> , 
	bError=> , 
	bBusy=> );
	// Kollar om något är knutet till inputen usiSpeed. Om inte körs ej detta block.	
	IF mSpeedEnableCheck(usiSpeed,usiOutput => usiOutput) THEN 
		fbReadWriteHoldingReg_usiSpeed(
		sIPAddr:= sIpAddr, 
		nTCPPort:= INT_TO_UINT(nTCPPort), 
		nUnitID:= INT_TO_BYTE(nUnitID), 
		mBusAdr:=4185 + offset, 
		bEnable:=bSekvensFlagga , 
		iWrite:=usiOutput , 
		iRead=> , 
		bError=> , 
		bBusy=> );
	END_IF;
	
	fbReadWriteHoldingRegSummerSetpoint(
	sIPAddr:= sIpAddr, 
	nTCPPort:= INT_TO_UINT(nTCPPort), 
	nUnitID:= INT_TO_BYTE(nUnitID), 
	mBusAdr:= 4141 + offset, 
	bEnable:= bSekvensFlagga, 
	iWrite:= fRealToWord(T1_SP,10), 
	iRead=> , 
	bError=> , 
	bBusy=> );
	
	fbReadWriteHoldingRegWinterSetpoint(
	sIPAddr:= sIpAddr, 
	nTCPPort:= INT_TO_UINT(nTCPPort), 
	nUnitID:= INT_TO_BYTE(nUnitID), 
	mBusAdr:= 4142 + offset, 
	bEnable:= bSekvensFlagga, 
	iWrite:= fRealToWord(T1_SP,10), 
	iRead=> , 
	bError=> , 
	bBusy=> );
	
//Communication error
	fbKommTof(IN:=FB_MBReadRegs_T1.bError , PT:=T#20S , Q=> , ET=> ); 
	fbKommTon(bInput:=fbKommTof.Q , tAlarmDelay:=T#20M , bAutoReset:= , bAlarmOutput=> );
	FAULT :=fbKommTon.bAlarmOutput;
		
//Write busy	
	oaksgvl.aBModbusBusyFlagga[iModbusLoop,nUnitID] := FB_MBReadRegs_T1.bBusy OR FB_MBReadRegs_T3.bBusy OR FB_MBReadRegs_MachineState.bBusy OR FB_MBReadRegs_Op.bBusy OR fbReadWriteHoldingReg_bStartStopp.bBusy OR fbReadWriteHoldingReg_usiSpeed.bBusy OR
	fbReadWriteHoldingRegSummerSetpoint.bBusy OR fbReadWriteHoldingRegWinterSetpoint.bBusy;

	
	fbHightempAlarm(
	bInput:= , 
	tAlarmDelay:= fRealToMinute(T1_HAD), 
	bAutoReset:= , 
	bAlarmOutput=>T1_HAL , 
	bEnable:= , 
	rProcessValue:=T1_PV , 
	rHighLimit:= T1_AHL);
	
	fbLowtempAlarm(
	bInput:= , 
	tAlarmDelay:= fRealToMinute(T1_LAD), 
	bAutoReset:= , 
	bAlarmOutput=>T1_LAL , 
	bEnable:= , 
	rProcessValue:=T1_PV , 
	rLowLimit:=T1_ALL );

METHOD PRIVATE mSpeedEnableCheck : BOOL // Blir TRUE om en USINT är knuten till ingången annars FALSE
VAR_INPUT
	usiTempToUse : ANY; //Kollar om det är en USINT knuten till ingången.
END_VAR
VAR
	pAnyUsint : POINTER TO USINT;
END_VAR
VAR_OUTPUT
	usiOutput : USINT; // Om en USINT är knuten till ingången följs denna annars alltid 0
END_VAR
//Temp select
IF usiTempToUse.TypeClass = __SYSTEM.TYPE_CLASS.TYPE_USINT THEN
	pAnyUsint := usiTempToUse.pValue;
	mSpeedEnableCheck := TRUE;
	usiOutput := pAnyUsint^;
ELSE
	mSpeedEnableCheck := FALSE;
	usiOutput := 0;
END_IF
END_METHOD

END_FUNCTION_BLOCK

// oaksModbusLibrary/Fidelix/FXIO (IO-kort)/Givarblock/fbFxIO_Sensor
//Givarblock för Fidelix AI8 (används med fbFx_AI8)
//OBS se manual för FXIO: https://oaksab.sharepoint.com/sites/Utveckling/_layouts/15/Doc.aspx?sourcedoc={22bc18e8-aa49-48c1-a1e6-a272a7cd26b5}&action=edit&wd=target%28Integrationer.one%7C5ac70296-2750-4373-ab29-5663253fae71%2FFxIO%20%28Fidelix%20IO-kort%5C%29%7C584643fa-d9bd-4007-939c-93e7e7825215%2F%29&wdorigin=703
FUNCTION_BLOCK fbFxIO_Sensor
VAR_INPUT
	nAIType			: BYTE := 0;		//Bygel på ingång: 0=(U) 0-10V, 1=(I) 0-25mA, 2=(T)emp
	rAISclRawMin	: REAL := 0;		//Min skalning för aktiv ingång i ingångsvärde (V eller mA)
	rAISclRawMax	: REAL := 10;		//Max skalning för aktiv ingång i ingångsvärde (V eller mA)
	rAISclEngMin	: REAL := 0;		//Min skalning för aktiv ingång i ingenjörsenhet
	rAISclEngMax	: REAL := 100;		//Max skalning för aktiv ingång i ingenjörsenhet
	nTempType		: BYTE := 0;		//Typ av passiv givare: 0=PT1000, 1=NI1000, 2=NI1000-LG, 3=NTC10, 4=TAC, 5=Egen (använd arUserTable)
	udiDamp			: UDINT := 0;		//Dämpning av givarvärde (sekunder)
	tAlarmDelay		: TIME := T#1S;		//Larmfördröjning givarfel (sekunder)
END_VAR

VAR_OUTPUT
	rPV 			: REAL;		//Givarvärde 
	FAULT AT %M* 	: BOOL;		//Givarfel ~wp:
END_VAR

VAR
	rRawIn : REAL;
	rRawUIn : REAL;
	rRawU_I : REAL;
	rRawOhm	: REAL;
	bFault	: BOOL;
	rPVint		: REAL;
	fbDamp	: Tc3_BA.FB_BA_TiAvrg;
	fbFault	: fbAlarm;											
END_VAR

VAR PERSISTENT
	//Fyll i X-led [n, 1]. Y-led är [n, 2] (justera vid behov)									  
	arUserTable	: ARRAY[1..20, 1..2] OF REAL := [		0	,	-40, 		 
		                                            	0	,	-30, 
                                                    	0	,	-20, 
                                                    	0	,	-10,
                                                    	0	,	0,
                                                    	0	,	10,
                                                   	 	0	,	20,
                                                    	0	,	25,
                                                    	0	,	30,
                                                    	0	,	40,
                                                    	0	,	50,
                                                   	 	0	,	60,
                                                    	0	,	70,
                                                    	0	,	80,
                                                    	0	,	90,
                                                    	0	,	100,
                                                    	0	,	110,
                                                    	0	,	120,
                                                    	0	,	130,
                                                    	0	,	140		];
END_VAR

rRawUIn := (rRawIn / 65535) * 10;	//Beräkna spänning på ingång som används för alla andra givartypsberäkningar

IF nAIType < 2 THEN			//Om 0-10V eller 0-25mA
	
	IF nAIType = 0 THEN			//Om 0-10V, använd råvärde i 0-10V
		rRawU_I := rRawUIn;
	ELSIF nAIType = 1 THEN		//Om 0-25mA, räkna om från 0-10V till 0-25mA
		rRawU_I := (rRawUIn) * 2.5;
	END_IF;	
	
	bFault := (rRawU_I < rAISclRawMin) OR (rRawU_I > rAISclRawMax);	//Givarfel om råvärde utanför angivet område
	rPVint := fScale2p(rX := rRawU_I, X1 := rAISclRawMin, X2 := rAISclRawMax, Y1 := rAISclEngMin, Y2 := rAISclEngMax);	//Beräkna PV linjärt enligt råvärde & ing.enhet min/max
ELSE						//Annars om Temp
	rRawOhm	:= (4700 * (rRawUIn * 0.25)) / MAX((2.5 - rRawUIn * 0.25), 0.000000000001);	//Beräkna ohm
	mGT();	//Kör metod som beräknar givarvärde och givarfel
END_IF

IF udiDamp > 0 THEN	//Dämpa givarvärde eller skriv det utan dämpning
	fbDamp(bEn := TRUE, rIn := rPVint, udiIntval_sec := 1, udiNumOfElem := udiDamp, rOut => rPV);
ELSE
	rPV := rPVint;
END_IF

fbFault(bInput := bFault, tAlarmDelay := tAlarmDelay, bAutoReset := TRUE, bAlarmOutput => FAULT);	//Givarfelslarm

METHOD PRIVATE mGT

VAR
	arUsed: ARRAY[1..20, 1..2] OF REAL;	

	arPT1000: ARRAY[1..20, 1..2] OF REAL := [	842.70	,	-40, 
												882.20	,	-30, 
												921.60	,	-20, 
												960.90	,	-10,
												1000  	,	0,
												1039  	,	10,
												1077.9	,	20,
												1097.4	,	25,
												1116.7	,	30,
												1155.4	,	40,
												1194  	,	50,
												1232.4	,	60,
												1270  	,	70,
												1308.9	,	80,
												1347  	,	90,
												1385  	,	100,
												1422  	,	110,
												1460.6	,	120,
												1498.2	,	130,
												1535.8	,	140		];
												
	arNI1000: ARRAY[1..20, 1..2] OF REAL := [	791.00	,	-40,   
												842.00	,	-30,   
												893.00	,	-20,   
												946.00	,	-10,   
												1000  	,	0,     
												1056  	,	10,    
												1112  	,	20,    
												1141  	,	25,    
												1171  	,	30,    
												1230  	,	40,    
												1291  	,	50,    
	                                            1353  	,	60,    
                                                1417  	,	70,    
                                                1483  	,	80,    
                                                1549  	,	90,    
                                                1618  	,	100,   
                                                1688  	,	110,   
                                                1760  	,	120,   
											    1853  	,	130,   
												1909  	,	140		];
												
												
												
	arNI1000LG: ARRAY[1..20, 1..2] OF REAL := [	830.83	 	,	-40,   
												871.69	 	,	-30,   
												913.48	 	,	-20,   
												956.24	 	,	-10,   
												1000	   	,	0,     
												1044.79		,	10,    
												1090.65		,	20,    
												1113.99		,	25,    
												1137.61		,	30,    
												1185.71		,	40,    
												1234.97		,	50,    
												1285.44		,	60,    
												1337.14		,	70,    
												1390.12		,	80,    
												1444.39		,	90,    
												1500	   	,	100,   
												1556.98		,	110,   
												1615.36		,	120,   
												1675.18		,	130,   
												1736.47		,	140		];
																							
	arNTC10: ARRAY[1..20, 1..2] OF REAL := [	0.23   		,	140,
												0.30   		,	130,
												0.39    	,	120,
												0.51    	,	110,
												0.68      	,	100,
			                                    0.92   		,	90 ,
                                                1.26   		,	80 ,
                                                1.75   		,	70 ,
                                                2.49    	,	60 ,
                                                3.60    	,	50 ,
                                                5.32    	,	40 ,
                                                8.06    	,	30 ,
                                                10.00   	,	25 ,
                                                12.49   	,	20 ,
                                                19.90   	,	10 ,
                                                32.65      	,	0  ,
                                                55.30   	,	-10,
                                                96.97   	,	-20,
                                                176.68  	,	-30,
                                                335.67  	,	-40		];
											
	arTAC: ARRAY[1..20, 1..2] OF REAL := 	[	77    	,	140,   
												95    	,	130,   
		                                        118   	,	120,   
                                                149   	,	110,   
                                                187     ,	100,   
                                                230  	,	90 ,   
                                                303  	,	80 ,   
                                                403  	,	70 ,   
                                                545  	,	60 ,   
                                                750  	,	50 ,   
                                                1049 	,	40 ,   
                                                1496 	,	30 ,   
                                                1801 	,	25 ,   
                                                2177 	,	20 ,   
                                                3241 	,	10 ,   
                                                4940    ,	0  ,   
                                                7730 	,	-10,   
                                                12443	,	-20,   
                                                20659	,	-30,   
                                                20659	,	-30		];
												
END_VAR
CASE THIS^.nTempType OF
	0:	arUsed := arPT1000;
	1:	arUsed := arNI1000;
	2:	arUsed := arNI1000LG;
	3:	arUsed := arNTC10;
	4:	arUsed := arTAC;
	5: 	arUsed := THIS^.arUserTable;
END_CASE

THIS^.bFault := (THIS^.rRawOhm > arUsed[20,1]) OR (THIS^.rRawOhm < arUsed[1,1]);

THIS^.rPVint := fScale20p(rX := THIS^.rRawOhm,
	X1	:=	arUsed[	1	,1],
	X2	:=	arUsed[	2	,1],
	X3	:=	arUsed[	3	,1],
	X4	:=	arUsed[	4	,1],
	X5	:=	arUsed[	5	,1],
	X6	:=	arUsed[	6	,1],
	X7	:=	arUsed[	7	,1],
	X8	:=	arUsed[	8	,1],
	X9	:=	arUsed[	9	,1],
	X10	:=	arUsed[	10	,1],
	X11	:=	arUsed[	11	,1],
	X12	:=	arUsed[	12	,1],
	X13	:=	arUsed[	13	,1],
	X14	:=	arUsed[	14	,1],
	X15	:=	arUsed[	15	,1],
	X16	:=	arUsed[	16	,1],
	X17	:=	arUsed[	17	,1],
	X18	:=	arUsed[	18	,1],
	X19	:=	arUsed[	19	,1],
	X20	:=	arUsed[	20	,1],
	Y1	:=	arUsed[	1	,2],
	Y2	:=	arUsed[	2	,2],
	Y3	:=	arUsed[	3	,2],
	Y4	:=	arUsed[	4	,2],
	Y5	:=	arUsed[	5	,2],
	Y6	:=	arUsed[	6	,2],
	Y7	:=	arUsed[	7	,2],
	Y8	:=	arUsed[	8	,2],
	Y9	:=	arUsed[	9	,2],
	Y10	:=	arUsed[	10	,2],
	Y11	:=	arUsed[	11	,2],
	Y12	:=	arUsed[	12	,2],
	Y13	:=	arUsed[	13	,2],
	Y14	:=	arUsed[	14	,2],
	Y15	:=	arUsed[	15	,2],
	Y16	:=	arUsed[	16	,2],
	Y17	:=	arUsed[	17	,2],
	Y18	:=	arUsed[	18	,2],
	Y19	:=	arUsed[	19	,2],
	Y20	:=	arUsed[	20	,2]	);
END_METHOD

METHOD PUBLIC mRaw : REAL
VAR_INPUT
	wRaw : WORD;
END_VAR
THIS^.rRawIn := wRaw;
END_METHOD

END_FUNCTION_BLOCK

// oaksModbusLibrary/Fidelix/FXIO (IO-kort)/Modulblock/fbFxIO_AI8
//Fidelix AI-8 IO-modul över ModbusTCP (används med t ex Moxa). Används med givarblock för fidelix, fbFxIO_Sensor
//Modulversion 1.x, funkar förhoppningsvis med senare versioner också
//Endast 16 bitars upplösning på AI i denna version, kan ökas till 20 bitar om det behövs
//Robert H, Oaks. 23-09-13
//Ver. 1.1 
//OBS se manual för FXIO: https://oaksab.sharepoint.com/sites/Utveckling/_layouts/15/Doc.aspx?sourcedoc={22bc18e8-aa49-48c1-a1e6-a272a7cd26b5}&action=edit&wd=target%28Integrationer.one%7C5ac70296-2750-4373-ab29-5663253fae71%2FFxIO%20%28Fidelix%20IO-kort%5C%29%7C584643fa-d9bd-4007-939c-93e7e7825215%2F%29&wdorigin=703
{attribute 'initialize_on_call'}
FUNCTION_BLOCK fbFxIO_AI8
VAR_INPUT
	bEnable 	: BOOL := TRUE; //Aktivering
	modbusTCP 	: ST_ModbusTCP;
	nUnitID		: BYTE := 0;
	tTimeOut 	: TIME := T#5S;	//Kom. timeout
	
	{attribute 'initialize_on_call'}
	rfbAI1 : REFERENCE TO fbFxIO_Sensor;	//Analog in-block 1
	
	{attribute 'initialize_on_call'}
	rfbAI2 : REFERENCE TO fbFxIO_Sensor;	//Analog in-block 2
	
	{attribute 'initialize_on_call'}
	rfbAI3 : REFERENCE TO fbFxIO_Sensor;	//Analog in-block 3
	
	{attribute 'initialize_on_call'}
	rfbAI4 : REFERENCE TO fbFxIO_Sensor;	//Analog in-block 4
	
	{attribute 'initialize_on_call'}
	rfbAI5 : REFERENCE TO fbFxIO_Sensor;	//Analog in-block 5
	
	{attribute 'initialize_on_call'}
	rfbAI6 : REFERENCE TO fbFxIO_Sensor;	//Analog in-block 6
	
	{attribute 'initialize_on_call'}
	rfbAI7 : REFERENCE TO fbFxIO_Sensor;	//Analog in-block 7
	
	{attribute 'initialize_on_call'}
	rfbAI8 : REFERENCE TO fbFxIO_Sensor;	//Analog in-block 8
END_VAR

VAR_OUTPUT
	sPV8 	: STRING;	//Modbus konfiguering
	bFAULT 	: BOOL;		//Kommunikationsfel
END_VAR

VAR
	sIP: STRING(255);
	sPort: STRING(255);
	sModbusID: STRING(255);
	sModbusLoop: STRING(255);
	sTemp : STRING(255);
	iStep: INT;
	bError: BOOL;
	bBusy: BOOL;	
	bSekvensFlagga : BOOL;
	
	FB_MBReadRegs_Values: FB_MBReadRegs;
	awReadRegs1 : ARRAY[0..7] OF WORD;
	
	FB_MBWriteRegs_AIused: FB_MBWriteSingleReg;
	wAIused : WORD;
	
	//Communication error
	fbKommTof : tof; 
	fbKommTon : fbAlarm;

	R_TRIG_Sekvens: R_TRIG;
	
END_VAR

IF nUnitID <> 0 THEN
	//Sekvens	
		R_TRIG_Sekvens(CLK:= oaksGVL.aBModbusSekvens[modbusTCP.iModbusLoop] = BYTE_TO_INT(nUnitID), Q=> bSekvensFlagga);
		
	//Modbus config
		sIP := CONCAT (modbusTCP.sIPAddr, '');
		sPort := CONCAT ('<br>Port: ', UINT_TO_STRING(modbusTCP.nTCPPort)); 								
		sModbusID := CONCAT('<br>ID: ', BYTE_TO_STRING(nUnitID));
		sModbusLoop := CONCAT('<br>Loop: ', INT_TO_STRING(modbusTCP.iModbusLoop));	
	
		sTemp := sIP;
		sTemp := CONCAT(sTemp, sPort);
		sTemp := CONCAT(sTemp, sModbusID);
		sTemp := CONCAT(sTemp, sModbusLoop);
		
		sPV8 := sTemp;
	
		CASE iStep OF
	
		0: 	//Start/reset
			bBusy := FALSE;
					
			IF bEnable AND bSekvensFlagga THEN
				iStep := 1;
				bError := FALSE;
			END_IF
			
		1: 	//Läs analogingångar
			bBusy := TRUE;
				
			FB_MBReadRegs_Values.bExecute := TRUE;
		
			FB_MBReadRegs_Values(
			sIPAddr:= modbusTCP.sIpAddr, 
			nTCPPort:= modbusTCP.nTCPPort, 
			nUnitID:= nUnitID, 
			nQuantity:= 8,
			nMBAddr:= 0, 
			cbLength:= SIZEOF(awReadRegs1), 
			pDestAddr:= ADR(awReadRegs1), 
			bExecute:= , 
			tTimeout:= tTimeOut, 
			bBusy=> , 
			bError=> , 
			nErrId=> , 
			cbRead=> );	
			
			//Error 
			IF FB_MBReadRegs_Values.bError THEN
				FB_MBReadRegs_Values(bExecute := FALSE);
				iStep := 99;
			END_IF
		
			//Läs råvärden och gå till nästa steg
			IF NOT FB_MBReadRegs_Values.bBusy AND NOT FB_MBReadRegs_Values.bError THEN
				
				mAI(rfbAI1, wRaw := awReadRegs1[0]);
				mAI(rfbAI2, wRaw := awReadRegs1[1]);
				mAI(rfbAI3, wRaw := awReadRegs1[2]);
				mAI(rfbAI4, wRaw := awReadRegs1[3]);
				mAI(rfbAI5, wRaw := awReadRegs1[4]);
				mAI(rfbAI6, wRaw := awReadRegs1[5]);
				mAI(rfbAI7, wRaw := awReadRegs1[6]);
				mAI(rfbAI8, wRaw := awReadRegs1[7]);
				
				FB_MBReadRegs_Values(bExecute := FALSE);
				bError := FALSE;
				iStep := 2;
			END_IF;
		
			
		2:	//Aktivera endast ingångar som används (för att öka prestanda på inläsning AI)
			wAIused.0 := __ISVALIDREF(rfbAI1);
			wAIused.1 := __ISVALIDREF(rfbAI2);
			wAIused.2 := __ISVALIDREF(rfbAI3);
			wAIused.3 := __ISVALIDREF(rfbAI4);
			wAIused.4 := __ISVALIDREF(rfbAI5);
			wAIused.5 := __ISVALIDREF(rfbAI6);
			wAIused.6 := __ISVALIDREF(rfbAI7);
			wAIused.7 := __ISVALIDREF(rfbAI8);
			
			FB_MBWriteRegs_AIused.bExecute := TRUE;
			
			FB_MBWriteRegs_AIused(
				sIPAddr:= modbusTCP.sIpAddr, 
				nTCPPort:= modbusTCP.nTCPPort, 
				nUnitID:= nUnitID,
				nMBAddr:= 10,
				nValue:= wAIused, 
				bExecute:= , 
				tTimeout:= tTimeout , 
				bBusy=> , 
				bError=> , 
				nErrId=> );
			
			//Error 
			IF FB_MBWriteRegs_AIused.bError THEN
				FB_MBWriteRegs_AIused(bExecute := FALSE);
				iStep := 99;
			END_IF
				
			//Gå till nästa steg	
			IF NOT FB_MBWriteRegs_AIused.bBusy AND NOT FB_MBWriteRegs_AIused.bError THEN
				
				FB_MBWriteRegs_AIused(bExecute := FALSE);
				bError := FALSE;
				iStep := 3;
			END_IF;
			
		3: //Done
			bBusy := FALSE;
			iStep := 0;
	
		99: //Error handling
			bBusy := FALSE;
			bError := TRUE;
			iStep := 0;
			
	END_CASE
		
	//Communication error
		fbKommTof(IN:=bError , PT:=T#20S , Q=> , ET=> );
		fbKommTon(bInput:=fbKommTof.Q , tAlarmDelay:=T#1M , bAutoReset:= , bAlarmOutput=> );
		bFAULT :=fbKommTon.bAlarmOutput;
			
	//Write busy	
		oaksgvl.aBModbusBusyFlagga[modbusTCP.iModbusLoop,nUnitID] := bBusy;
ELSE
	bFAULT := TRUE;
END_IF

METHOD PRIVATE mAI
VAR_INPUT
	refFidelixAI : REFERENCE TO fbFxIO_Sensor;
	wRaw : WORD;
END_VAR
IF __ISVALIDREF(refFidelixAI) THEN		//Om AI-block används för ingång
	refFidelixAI.mRaw(wRaw);			//Skicka över råvärde
END_IF;
END_METHOD

END_FUNCTION_BLOCK

// oaksModbusLibrary/Fidelix/FXIO (IO-kort)/Modulblock/fbFxIO_AO8
//Fidelix AO-8 IO-modul över ModbusTCP (används med t ex Moxa)
//Modulversion 1.10 / 2.20, funkar förhoppningsvis med senare versioner också
//Skrivning av AO, samt skrivning av fallback-konfiguration för AO. Om fallback för AO är till (rAOxfallback > 0) aktiveras det i modulen då ingen kommunikation skett efter 30 sekunder
//Robert H, Oaks. 23-09-20
//Ver. 1.1
//OBS se manual för FXIO: https://oaksab.sharepoint.com/sites/Utveckling/_layouts/15/Doc.aspx?sourcedoc={22bc18e8-aa49-48c1-a1e6-a272a7cd26b5}&action=edit&wd=target%28Integrationer.one%7C5ac70296-2750-4373-ab29-5663253fae71%2FFxIO%20%28Fidelix%20IO-kort%5C%29%7C584643fa-d9bd-4007-939c-93e7e7825215%2F%29&wdorigin=703
FUNCTION_BLOCK fbFxIO_AO8
VAR_INPUT
	bEnable 	: BOOL := TRUE; //Aktivering
	modbusTCP 	: ST_ModbusTCP;
	nUnitID		: BYTE := 0;
	tTimeOut 	: TIME :=T#5S;
	bSetConfig	: BOOL := FALSE; //Skriv fallback-konfiguration
	
	{attribute 'initialize_on_call'}
	rrAO1 		 : REFERENCE TO REAL; //Analog ut 1 (0-100%)
	rAO1fallback : REAL := -1; //Fallback (0-100%, sätt till -1 för ej fallback!)
	{attribute 'initialize_on_call'}
	rrAO2 		 : REFERENCE TO REAL; //Analog ut 2 (0-100%)
	rAO2fallback : REAL := -1; //Fallback (0-100%, sätt till -1 för ej fallback!)
	{attribute 'initialize_on_call'}
	rrAO3 		 : REFERENCE TO REAL; //Analog ut 3 (0-100%)
	rAO3fallback : REAL := -1; //Fallback (0-100%, sätt till -1 för ej fallback!)
	{attribute 'initialize_on_call'}
	rrAO4 		 : REFERENCE TO REAL; //Analog ut 4 (0-100%)
	rAO4fallback : REAL := -1; //Fallback (0-100%, sätt till -1 för ej fallback!)
	{attribute 'initialize_on_call'}
	rrAO5 		 : REFERENCE TO REAL; //Analog ut 5 (0-100%)
	rAO5fallback : REAL := -1; //Fallback (0-100%, sätt till -1 för ej fallback!)
	{attribute 'initialize_on_call'}
	rrAO6 		 : REFERENCE TO REAL; //Analog ut 6 (0-100%)
	rAO6fallback : REAL := -1; //Fallback (0-100%, sätt till -1 för ej fallback!)
	{attribute 'initialize_on_call'}
	rrAO7 		 : REFERENCE TO REAL; //Analog ut 7 (0-100%)
	rAO7fallback : REAL := -1; //Fallback (0-100%, sätt till -1 för ej fallback!)
	{attribute 'initialize_on_call'}
	rrAO8 		 : REFERENCE TO REAL; //Analog ut 8 (0-100%)
	rAO8fallback : INT := -1; //Fallback (0-100%, sätt till -1 för ej fallback!)
	
END_VAR
	
VAR_OUTPUT
	sPV8 	: STRING;	//Modbus konfiguering
	bFAULT 	: BOOL;		//Kommunikationsfel
END_VAR

VAR
	sIP: STRING(255);
	sPort: STRING(255);
	sModbusID: STRING(255);
	sModbusLoop: STRING(255);
	sTemp : STRING(255);	

	bSekvensFlagga : BOOL;
	iStep: INT;
	bError: BOOL;
	bBusy: BOOL;
	
	FB_MBWriteRegs_Fallback: FB_MBWriteRegs;
	wFallback : ARRAY[1..8] OF WORD; 
	
	FB_MBWriteRegs_AO: FB_MBWriteRegs;
	wAO : ARRAY[1..8] OF WORD;

	//Communication error
	fbKommTof : tof; 
	fbKommTon : fbAlarm;
		
	R_TRIG_Sekvens: R_TRIG;
END_VAR

//Sekvens	
	R_TRIG_Sekvens(CLK:= oaksGVL.aBModbusSekvens[modbusTCP.iModbusLoop] = BYTE_TO_INT(nUnitID), Q=> bSekvensFlagga);
	
	
//Modbus config
	sIP := CONCAT (modbusTCP.sIPAddr, '');
	sPort := CONCAT ('<br>Port: ', UINT_TO_STRING(modbusTCP.nTCPPort)); 								
	sModbusID := CONCAT('<br>ID: ', BYTE_TO_STRING(nUnitID));
	sModbusLoop := CONCAT('<br>Loop: ', INT_TO_STRING(modbusTCP.iModbusLoop));	

	sTemp := sIP;
	sTemp := CONCAT(sTemp, sPort);
	sTemp := CONCAT(sTemp, sModbusID);
	sTemp := CONCAT(sTemp, sModbusLoop);
	
	sPV8 := sTemp;

	CASE iStep OF

	0: 	//Start/reset
		bBusy := FALSE;

		IF bEnable AND bSekvensFlagga THEN
			iStep := 1;
			bError := FALSE;
		END_IF

	1:	//Skriv fallbackvärden
		wFallback[1] := SEL(rAO1fallback < 0, REAL_TO_WORD((1023 * (rAO1fallback / 100))) OR 16#8000, 0);
		wFallback[2] := SEL(rAO2fallback < 0, REAL_TO_WORD((1023 * (rAO2fallback / 100))) OR 16#8000, 0);
		wFallback[3] := SEL(rAO3fallback < 0, REAL_TO_WORD((1023 * (rAO3fallback / 100))) OR 16#8000, 0);
		wFallback[4] := SEL(rAO4fallback < 0, REAL_TO_WORD((1023 * (rAO4fallback / 100))) OR 16#8000, 0);
		wFallback[5] := SEL(rAO5fallback < 0, REAL_TO_WORD((1023 * (rAO5fallback / 100))) OR 16#8000, 0);
		wFallback[6] := SEL(rAO6fallback < 0, REAL_TO_WORD((1023 * (rAO6fallback / 100))) OR 16#8000, 0);
		wFallback[7] := SEL(rAO7fallback < 0, REAL_TO_WORD((1023 * (rAO7fallback / 100))) OR 16#8000, 0);
		wFallback[8] := SEL(rAO8fallback < 0, REAL_TO_WORD((1023 * (rAO8fallback / 100))) OR 16#8000, 0);
			
		IF bSetConfig THEN
			FB_MBWriteRegs_Fallback.bExecute := TRUE;
			bBusy := TRUE;
		END_IF
			
		FB_MBWriteRegs_Fallback(
		sIPAddr:= modbusTCP.sIpAddr, 
		nTCPPort:= modbusTCP.nTCPPort, 
		nUnitID:= nUnitID, 
		nQuantity:= 8, 
		nMBAddr:= 9, 
		cbLength:= SIZEOF(wFallback), 
		pSrcAddr:= ADR(wFallback), 
		bExecute:=, 
		tTimeout:= tTimeOut, 
		bBusy=> , 
		bError=> , 
		nErrId=> );
		
		IF FB_MBWriteRegs_Fallback.bError THEN
			FB_MBWriteRegs_Fallback(bExecute := FALSE);
			iStep := 99;
		END_IF
	
		//Next step
		IF NOT FB_MBWriteRegs_Fallback.bBusy AND NOT FB_MBWriteRegs_Fallback.bError THEN
			FB_MBWriteRegs_Fallback(bExecute := FALSE);
			bSetConfig := FALSE; 
			bError := FALSE;
			iStep := 2;
		END_IF;

	2: //Write outputs
		bBusy := TRUE;	
			
		IF __ISVALIDREF(rrAO1) THEN wAO[1] := MAX(0, MIN(1023, REAL_TO_WORD(1023 * (rrAO1 / 100)))); END_IF
		IF __ISVALIDREF(rrAO2) THEN wAO[2] := MAX(0, MIN(1023, REAL_TO_WORD(1023 * (rrAO2 / 100)))); END_IF	
		IF __ISVALIDREF(rrAO3) THEN wAO[3] := MAX(0, MIN(1023, REAL_TO_WORD(1023 * (rrAO3 / 100)))); END_IF
		IF __ISVALIDREF(rrAO4) THEN wAO[4] := MAX(0, MIN(1023, REAL_TO_WORD(1023 * (rrAO4 / 100)))); END_IF
		IF __ISVALIDREF(rrAO5) THEN wAO[5] := MAX(0, MIN(1023, REAL_TO_WORD(1023 * (rrAO5 / 100)))); END_IF
		IF __ISVALIDREF(rrAO6) THEN wAO[6] := MAX(0, MIN(1023, REAL_TO_WORD(1023 * (rrAO6 / 100)))); END_IF
		IF __ISVALIDREF(rrAO7) THEN wAO[7] := MAX(0, MIN(1023, REAL_TO_WORD(1023 * (rrAO7 / 100)))); END_IF
		IF __ISVALIDREF(rrAO8) THEN wAO[8] := MAX(0, MIN(1023, REAL_TO_WORD(1023 * (rrAO8 / 100)))); END_IF
		
		FB_MBWriteRegs_AO.bExecute := TRUE;
		
		FB_MBWriteRegs_AO(
		sIPAddr:= modbusTCP.sIpAddr, 
		nTCPPort:= modbusTCP.nTCPPort, 
		nUnitID:= nUnitID, 
		nQuantity:= 8, 
		nMBAddr:= 0, 
		cbLength:= SIZEOF(wAO), 
		pSrcAddr:= ADR(wAO), 
		bExecute:=, 
		tTimeout:= tTimeOut, 
		bBusy=> , 
		bError=> , 
		nErrId=> );
		
		IF FB_MBWriteRegs_AO.bError THEN
			FB_MBWriteRegs_AO(bExecute := FALSE);
			iStep := 99;
		END_IF
	
		//Next step
		IF NOT FB_MBWriteRegs_AO.bBusy AND NOT FB_MBWriteRegs_AO.bError THEN
			FB_MBWriteRegs_AO(bExecute := FALSE);
			bError := FALSE;
			iStep := 20;
		END_IF;

	20: //Done
		bBusy := FALSE;
		iStep := 0;

	99: //Error handling
		bBusy := FALSE;
		bError := TRUE;
		iStep := 0;
		
END_CASE

//Communication error
	fbKommTof(IN:=bError , PT:=T#20S , Q=> , ET=> );
	fbKommTon(bInput:=fbKommTof.Q , tAlarmDelay:=T#1M , bAutoReset:= , bAlarmOutput=> );
	bFAULT :=fbKommTon.bAlarmOutput;
		
//Write busy	
	oaksgvl.aBModbusBusyFlagga[modbusTCP.iModbusLoop,nUnitID] := bBusy;

END_FUNCTION_BLOCK

// oaksModbusLibrary/Fidelix/FXIO (IO-kort)/Modulblock/fbFxIO_Combi36
//Fidelix Combi-36 IO-modul över ModbusTCP (används med t ex Moxa)
//Modulversion 1.10 / 2.20, funkar förhoppningsvis med senare versioner också
//Blocket kör underblock för alla separata moduler. nUnitID ska vara kortets startadress (följande moduler får startadress +1, +2 och +3)
//Robert H, Oaks. 23-09-20
//Ver. 1.1
//OBS se manual för FXIO: https://oaksab.sharepoint.com/sites/Utveckling/_layouts/15/Doc.aspx?sourcedoc={22bc18e8-aa49-48c1-a1e6-a272a7cd26b5}&action=edit&wd=target%28Integrationer.one%7C5ac70296-2750-4373-ab29-5663253fae71%2FFxIO%20%28Fidelix%20IO-kort%5C%29%7C584643fa-d9bd-4007-939c-93e7e7825215%2F%29&wdorigin=703

{attribute 'initialize_on_call'}
FUNCTION_BLOCK fbFxIO_Combi36
VAR_INPUT
	bEnable 	: BOOL := TRUE; //Aktivering
	modbusTCP 	: ST_ModbusTCP;	//Modbus-konfiguration
	nUnitID		: BYTE := 0;	//Moduladress
	tTimeOut 	: TIME := T#5S;	//Kom. timeout
	bBlink		: BOOL := FALSE;//Blinka lysdioder på kortet (för fysisk identifiering)
	bSetConfig	: BOOL := FALSE;//Skriv fallback-inställningar till modul (DO & AO)
	
	{attribute 'initialize_on_call'}
	rbDI1 : REFERENCE TO BOOL;//Digitalingång 1
	{attribute 'initialize_on_call'}
	rbDI2 : REFERENCE TO BOOL;//Digitalingång 2
	{attribute 'initialize_on_call'}
	rbDI3 : REFERENCE TO BOOL;//Digitalingång 3
	{attribute 'initialize_on_call'}
	rbDI4 : REFERENCE TO BOOL;//Digitalingång 4
	{attribute 'initialize_on_call'}
	rbDI5 : REFERENCE TO BOOL;//Digitalingång 5
	{attribute 'initialize_on_call'}
	rbDI6 : REFERENCE TO BOOL;//Digitalingång 6
	{attribute 'initialize_on_call'}
	rbDI7 : REFERENCE TO BOOL;//Digitalingång 7
	{attribute 'initialize_on_call'}
	rbDI8 : REFERENCE TO BOOL;//Digitalingång 8
	{attribute 'initialize_on_call'}
	rbDI9 : REFERENCE TO BOOL;//Digitalingång 9
	{attribute 'initialize_on_call'}
	rbDI10 : REFERENCE TO BOOL;//Digitalingång 10
	{attribute 'initialize_on_call'}
	rbDI11 : REFERENCE TO BOOL;//Digitalingång 11
	{attribute 'initialize_on_call'}
	rbDI12 : REFERENCE TO BOOL;//Digitalingång 12
	
	{attribute 'initialize_on_call'}
	rbDO1 : REFERENCE TO BOOL;		//Digitalutgång 1
	nDO1fallback : BYTE := 0; 		//Fallback (0=Ej fallback, 1=Fallback 0, 2=Fallback 1);
	{attribute 'initialize_on_call'}
	rbDO2 : REFERENCE TO BOOL; 		//Digitalutgång 2
	nDO2fallback : BYTE := 0; 		//Fallback (0=Ej fallback, 1=Fallback 0, 2=Fallback 1);
	{attribute 'initialize_on_call'}
	rbDO3 : REFERENCE TO BOOL; 		//Digitalutgång 3
	nDO3fallback : BYTE := 0; 		//Fallback (0=Ej fallback, 1=Fallback 0, 2=Fallback 1);
	{attribute 'initialize_on_call'}
	rbDO4 : REFERENCE TO BOOL; 		//Digitalutgång 4
	nDO4fallback : BYTE := 0; 		//Fallback (0=Ej fallback, 1=Fallback 0, 2=Fallback 1);
	{attribute 'initialize_on_call'}
	rbDO5 : REFERENCE TO BOOL;		//Digitalutgång 5
	nDO5fallback : BYTE := 0; 		//Fallback (0=Ej fallback, 1=Fallback 0, 2=Fallback 1);
	{attribute 'initialize_on_call'}
	rbDO6 : REFERENCE TO BOOL;		//Digitalutgång 6
	nDO6fallback : BYTE := 0; 		//Fallback (0=Ej fallback, 1=Fallback 0, 2=Fallback 1);
	{attribute 'initialize_on_call'}
	rbDO7 : REFERENCE TO BOOL; 		//Digitalutgång 7
	nDO7fallback : BYTE := 0; 		//Fallback (0=Ej fallback, 1=Fallback 0, 2=Fallback 1);
	{attribute 'initialize_on_call'}
	rbDO8 : REFERENCE TO BOOL; 		//Digitalutgång 8
	nDO8fallback : BYTE := 0; 		//Fallback (0=Ej fallback, 1=Fallback 0, 2=Fallback 1);
	
	{attribute 'initialize_on_call'}
	rfbAI1 : REFERENCE TO fbFxIO_Sensor;	//Analog in-block 1
	{attribute 'initialize_on_call'}
	rfbAI2 : REFERENCE TO fbFxIO_Sensor;	//Analog in-block 2
	{attribute 'initialize_on_call'}	
	rfbAI3 : REFERENCE TO fbFxIO_Sensor;	//Analog in-block 3
	{attribute 'initialize_on_call'}
	rfbAI4 : REFERENCE TO fbFxIO_Sensor;	//Analog in-block 4
	{attribute 'initialize_on_call'}
	rfbAI5 : REFERENCE TO fbFxIO_Sensor;	//Analog in-block 5
	{attribute 'initialize_on_call'}
	rfbAI6 : REFERENCE TO fbFxIO_Sensor;	//Analog in-block 6
	{attribute 'initialize_on_call'}
	rfbAI7 : REFERENCE TO fbFxIO_Sensor;	//Analog in-block 7
	{attribute 'initialize_on_call'}
	rfbAI8 : REFERENCE TO fbFxIO_Sensor;	//Analog in-block 8
	
	{attribute 'initialize_on_call'}
	rrAO1 		 : REFERENCE TO REAL; //Analog ut 1 (0-100%)
	rAO1fallback : REAL := -1; //Fallback (0-100%, sätt till -1 för ej fallback!)
	{attribute 'initialize_on_call'}
	rrAO2 		 : REFERENCE TO REAL; //Analog ut 2 (0-100%)
	rAO2fallback : REAL := -1; //Fallback (0-100%, sätt till -1 för ej fallback!)
	{attribute 'initialize_on_call'}
	rrAO3 		 : REFERENCE TO REAL; //Analog ut 3 (0-100%)
	rAO3fallback : REAL := -1; //Fallback (0-100%, sätt till -1 för ej fallback!)
	{attribute 'initialize_on_call'}
	rrAO4 		 : REFERENCE TO REAL; //Analog ut 4 (0-100%)
	rAO4fallback : REAL := -1; //Fallback (0-100%, sätt till -1 för ej fallback!)
	{attribute 'initialize_on_call'}
	rrAO5 		 : REFERENCE TO REAL; //Analog ut 5 (0-100%)
	rAO5fallback : REAL := -1; //Fallback (0-100%, sätt till -1 för ej fallback!)
	{attribute 'initialize_on_call'}
	rrAO6 		 : REFERENCE TO REAL; //Analog ut 6 (0-100%)
	rAO6fallback : REAL := -1; //Fallback (0-100%, sätt till -1 för ej fallback!)
	{attribute 'initialize_on_call'}
	rrAO7 		 : REFERENCE TO REAL; //Analog ut 7 (0-100%)
	rAO7fallback : REAL := -1; //Fallback (0-100%, sätt till -1 för ej fallback!)
	{attribute 'initialize_on_call'}
	rrAO8 		 : REFERENCE TO REAL; //Analog ut 8 (0-100%)
	rAO8fallback : INT := -1; //Fallback (0-100%, sätt till -1 för ej fallback!)
	
END_VAR
VAR_OUTPUT
	sPV8 	: STRING;	//Modbus konfiguering
	bFAULT 	: BOOL;		//Kommunikationsfel
END_VAR
VAR
	fbSetConfigEdge : fbEdge;	

	fbM1	: fbFxIO_DI16;
	fbM2	: fbFxIO_DO8;
	fbM3	: fbFxIO_AI8; 
	fbM4	: fbFxIO_AO8;
END_VAR

fbSetConfigEdge(anyInput := bSetConfig, bIncr := TRUE);

IF bSetConfig THEN
	fbM2.bSetConfig := TRUE;
	fbM4.bSetConfig := TRUE;
END_IF

//Modul 1, DI16 (endast 12 ingångar finns på C36). Första adress
	fbM1.rbDI1 REF= rbDI1;
	fbM1.rbDI2 REF= rbDI2;
	fbM1.rbDI3 REF= rbDI3;
	fbM1.rbDI4 REF= rbDI4;
	fbM1.rbDI5 REF= rbDI5;
	fbM1.rbDI6 REF= rbDI6;
	fbM1.rbDI7 REF= rbDI7;
	fbM1.rbDI8 REF= rbDI8;
	fbM1.rbDI9 REF= rbDI9;
	fbM1.rbDI10 REF= rbDI10;
	fbM1.rbDI11 REF= rbDI11;
	fbM1.rbDI12 REF= rbDI12;
	fbM1(bEnable := bEnable, modbusTCP := modbusTCP, nUnitID := nUnitID, tTimeOut := tTimeOut, bBlink := bBlink);

	//Modbus-konfiguration och kom.larm från modul 1
	sPV8 := fbM1.sPV8;
	bFAULT := fbM1.bFAULT;

	//Modul 2, DO8. Andra adress
	fbM2.rbDO1 REF= rbDO1;
	fbM2.nDO1fallback := nDO1fallback;
	fbM2.rbDO2 REF= rbDO2;
	fbM2.nDO2fallback := nDO2fallback;
	fbM2.rbDO3 REF= rbDO3;
	fbM2.nDO3fallback := nDO3fallback;
	fbM2.rbDO4 REF= rbDO4;
	fbM2.nDO4fallback := nDO4fallback;
	fbM2.rbDO5 REF= rbDO5;
	fbM2.nDO5fallback := nDO5fallback;
	fbM2.rbDO6 REF= rbDO6;
	fbM2.nDO6fallback := nDO6fallback;
	fbM2.rbDO7 REF= rbDO7;
	fbM2.nDO7fallback := nDO7fallback;
	fbM2.rbDO8 REF= rbDO8;
	fbM2.nDO8fallback := nDO8fallback;
	fbM2(bEnable := bEnable, modbusTCP := modbusTCP, nUnitID := nUnitID + 1, tTimeOut := tTimeOut);
	
//Modul 3, AI8. Tredje adress
	fbM3.rfbAI1 REF= rfbAI1;
	fbM3.rfbAI2 REF= rfbAI2;
	fbM3.rfbAI3 REF= rfbAI3;
	fbM3.rfbAI4 REF= rfbAI4;
	fbM3.rfbAI5 REF= rfbAI5;
	fbM3.rfbAI6 REF= rfbAI6;
	fbM3.rfbAI7 REF= rfbAI7;
	fbM3.rfbAI8 REF= rfbAI8;
	fbM3(bEnable := bEnable, modbusTCP := modbusTCP, nUnitID := nUnitID + 2, tTimeOut := tTimeOut);
	
//Modul 4, AO8. Fjärde adress
	fbM4.rrAO1 REF= rrAO1;
	fbM4.rAO1fallback := rAO1fallback;
	fbM4.rrAO2 REF= rrAO2;
	fbM4.rAO2fallback := rAO2fallback;
	fbM4.rrAO3 REF= rrAO3;
	fbM4.rAO3fallback := rAO3fallback;
	fbM4.rrAO4 REF= rrAO4;
	fbM4.rAO4fallback := rAO4fallback;
	fbM4.rrAO5 REF= rrAO5;
	fbM4.rAO5fallback := rAO5fallback;
	fbM4.rrAO6 REF= rrAO6;
	fbM4.rAO6fallback := rAO6fallback;
	fbM4.rrAO7 REF= rrAO7;
	fbM4.rAO7fallback := rAO7fallback;
	fbM4.rrAO8 REF= rrAO8;
	fbM4.rAO8fallback := rAO8fallback;
	fbM4(bEnable := bEnable, modbusTCP := modbusTCP, nUnitID := nUnitID + 3, tTimeOut := tTimeOut);

bSetConfig := FALSE;

END_FUNCTION_BLOCK

// oaksModbusLibrary/Fidelix/FXIO (IO-kort)/Modulblock/fbFxIO_DI16
//Fidelix DI-16 IO-modul över ModbusTCP (används med t ex Moxa)
//Modulversion 1.10, funkar förhoppningsvis med senare versioner också
//Endast inläsning av DI i denna version. Konfiguration och inläsning av pulsräknare kan göras i framtiden vid behov.
//Robert H, Oaks. 23-09-12
//Ver. 1.1
//OBS se manual för FXIO: https://oaksab.sharepoint.com/sites/Utveckling/_layouts/15/Doc.aspx?sourcedoc={22bc18e8-aa49-48c1-a1e6-a272a7cd26b5}&action=edit&wd=target%28Integrationer.one%7C5ac70296-2750-4373-ab29-5663253fae71%2FFxIO%20%28Fidelix%20IO-kort%5C%29%7C584643fa-d9bd-4007-939c-93e7e7825215%2F%29&wdorigin=703
{attribute 'initialize_on_call'}
FUNCTION_BLOCK fbFxIO_DI16
VAR_INPUT
	bEnable 	: BOOL := TRUE; //Aktivering
	modbusTCP 	: ST_ModbusTCP;	//Modbus-konfiguration
	nUnitID		: BYTE := 0;	//Moduladress
	tTimeOut 	: TIME := T#5S;	//Kom. timeout
	bBlink		: BOOL := FALSE;//Blinka lysdioder på kortet (för fysisk identifiering)
	
	{attribute 'initialize_on_call'}
	rbDI1 : REFERENCE TO BOOL;//Digitalingång 1
	{attribute 'initialize_on_call'}
	rbDI2 : REFERENCE TO BOOL;//Digitalingång 2
	{attribute 'initialize_on_call'}
	rbDI3 : REFERENCE TO BOOL;//Digitalingång 3
	{attribute 'initialize_on_call'}
	rbDI4 : REFERENCE TO BOOL;//Digitalingång 4
	{attribute 'initialize_on_call'}
	rbDI5 : REFERENCE TO BOOL;//Digitalingång 5
	{attribute 'initialize_on_call'}
	rbDI6 : REFERENCE TO BOOL;//Digitalingång 6
	{attribute 'initialize_on_call'}
	rbDI7 : REFERENCE TO BOOL;//Digitalingång 7
	{attribute 'initialize_on_call'}
	rbDI8 : REFERENCE TO BOOL;//Digitalingång 8
	{attribute 'initialize_on_call'}
	rbDI9 : REFERENCE TO BOOL;//Digitalingång 9
	{attribute 'initialize_on_call'}
	rbDI10 : REFERENCE TO BOOL;//Digitalingång 10
	{attribute 'initialize_on_call'}
	rbDI11 : REFERENCE TO BOOL;//Digitalingång 11
	{attribute 'initialize_on_call'}
	rbDI12 : REFERENCE TO BOOL;//Digitalingång 12
	{attribute 'initialize_on_call'}
	rbDI13 : REFERENCE TO BOOL;//Digitalingång 13
	{attribute 'initialize_on_call'}
	rbDI14 : REFERENCE TO BOOL;//Digitalingång 14
	{attribute 'initialize_on_call'}
	rbDI15 : REFERENCE TO BOOL;//Digitalingång 15
	{attribute 'initialize_on_call'}
	rbDI16 : REFERENCE TO BOOL;//Digitalingång 16
END_VAR
VAR_OUTPUT
	
	sPV8 	: STRING;	//Modbus konfiguering
	bFAULT 	: BOOL;		//Kommunikationsfel
	
END_VAR
VAR
	sIP: STRING(255);
	sPort: STRING(255);
	sModbusID: STRING(255);
	sModbusLoop: STRING(255);
	sTemp : STRING(255);
	bSekvensFlagga : BOOL;
	
	iStep: INT;
	
	FB_MBReadRegs_InputRegs1: FB_MBReadRegs;
	wInputRegs1 : WORD; 
	
	FB_MBWriteRegs_Blink: FB_MBWriteSingleReg;
		
	//Communication error
	fbKommTof : tof; 
	fbKommTon : fbAlarm;

	R_TRIG_Sekvens: R_TRIG;
	
	fbEdge1 : fbEdge;
	
	bError : BOOL;
	bBusy : BOOL;
END_VAR

IF nUnitID <> 0 THEN
	//Sekvens	
		R_TRIG_Sekvens(CLK:= oaksGVL.aBModbusSekvens[modbusTCP.iModbusLoop] = BYTE_TO_INT(nUnitID), Q=> bSekvensFlagga);
		
	//Modbus config
		sIP := CONCAT (modbusTCP.sIPAddr, '');
		sPort := CONCAT ('<br>Port: ', UINT_TO_STRING(modbusTCP.nTCPPort)); 								
		sModbusID := CONCAT('<br>ID: ', BYTE_TO_STRING(nUnitID));
		sModbusLoop := CONCAT('<br>Loop: ', INT_TO_STRING(modbusTCP.iModbusLoop));	
	
		sTemp := sIP;
		sTemp := CONCAT(sTemp, sPort);
		sTemp := CONCAT(sTemp, sModbusID);
		sTemp := CONCAT(sTemp, sModbusLoop);
		
		sPV8 := sTemp;
		
	
	CASE iStep OF
	0:	// Start/reset
		bBusy := FALSE;
							
		IF bEnable AND bSekvensFlagga THEN
			iStep := 1;
			bError := FALSE;
		END_IF
		
	1:	//Läs digitala ingångar
		FB_MBReadRegs_InputRegs1(
			sIPAddr:= modbusTCP.sIpAddr, 
			nTCPPort:= modbusTCP.nTCPPort, 
			nUnitID:= nUnitID, 
			nQuantity:= 1, 
			nMBAddr:= 0, 
			cbLength:= SIZEOF(wInputRegs1), 
			pDestAddr:= ADR(wInputRegs1), 
			bExecute:= TRUE, 
			tTimeout:= tTimeOut, 
			bBusy=> , 
			bError=> , 
			nErrId=> , 
			cbRead=> );
			
		IF FB_MBReadRegs_InputRegs1.bError THEN
			FB_MBReadRegs_InputRegs1(bExecute := FALSE);
			iStep := 99;
		END_IF
		
		IF NOT FB_MBReadRegs_InputRegs1.bBusy AND NOT FB_MBReadRegs_InputRegs1.bError THEN
			FB_MBReadRegs_InputRegs1(bExecute := FALSE);
			bError := FALSE;
			iStep := 2;
		END_IF;	
		
	2:	//Överför till variabler
		IF __ISVALIDREF(rbDI1) THEN rbDI1 := NOT wInputRegs1.0; END_IF;
		IF __ISVALIDREF(rbDI2) THEN rbDI2 := NOT wInputRegs1.1; END_IF;
		IF __ISVALIDREF(rbDI3) THEN rbDI3 := NOT wInputRegs1.2; END_IF;
		IF __ISVALIDREF(rbDI4) THEN rbDI4 := NOT wInputRegs1.3; END_IF;
		IF __ISVALIDREF(rbDI5) THEN rbDI5 := NOT wInputRegs1.4; END_IF;
		IF __ISVALIDREF(rbDI6) THEN rbDI6 := NOT wInputRegs1.5; END_IF;
		IF __ISVALIDREF(rbDI7) THEN rbDI7 := NOT wInputRegs1.6; END_IF;
		IF __ISVALIDREF(rbDI8) THEN rbDI8 := NOT wInputRegs1.7; END_IF;
		IF __ISVALIDREF(rbDI9) THEN rbDI9 := NOT wInputRegs1.8; END_IF;
		IF __ISVALIDREF(rbDI10) THEN rbDI10 := NOT wInputRegs1.9; END_IF;
		IF __ISVALIDREF(rbDI11) THEN rbDI11 := NOT wInputRegs1.10; END_IF;
		IF __ISVALIDREF(rbDI12) THEN rbDI12 := NOT wInputRegs1.11; END_IF;
		IF __ISVALIDREF(rbDI13) THEN rbDI13 := NOT wInputRegs1.12; END_IF;
		IF __ISVALIDREF(rbDI14) THEN rbDI14 := NOT wInputRegs1.13; END_IF;
		IF __ISVALIDREF(rbDI15) THEN rbDI15 := NOT wInputRegs1.14; END_IF;
		IF __ISVALIDREF(rbDI16) THEN rbDI16 := NOT wInputRegs1.15; END_IF;
		
		iStep := 3;
		
	3:	//Skriv blinkfunktion
		fbEdge1(anyInput := bBlink);
		
		FB_MBWriteRegs_Blink(
				sIPAddr:= modbusTCP.sIpAddr, 
				nTCPPort:= modbusTCP.nTCPPort, 
				nUnitID:= nUnitID,
				nMBAddr:= 5,
				nValue:= 16#FFFF * BOOL_TO_UINT(bBlink), 
				bExecute:= fbEdge1.bEdgeSR, 
				tTimeout:= tTimeout , 
				bBusy=> , 
				bError=> , 
				nErrId=> );
		
		IF FB_MBWriteRegs_Blink.bError THEN
			FB_MBWriteRegs_Blink(bExecute := FALSE);
			iStep := 99;
		END_IF
		
		IF NOT FB_MBWriteRegs_Blink.bBusy AND NOT FB_MBWriteRegs_Blink.bError THEN
			FB_MBWriteRegs_Blink(bExecute := FALSE);
			bError := FALSE;
			fbEdge1(bRst := TRUE); 
			iStep := 20;
		END_IF;
			
		20: //Done
			bBusy := FALSE;
			iStep := 0;
		
		99: //Error handling
			bBusy := FALSE;
			bError := TRUE;
			iStep := 0;
			
		END_CASE;
		
	//Kommunikationsfel modul
		fbKommTof(IN:=bError , PT:=T#20S , Q=> , ET=> );
		fbKommTon(bInput:=fbKommTof.Q , tAlarmDelay:=T#1M , bAutoReset:= , bAlarmOutput=> );
		bFAULT :=fbKommTon.bAlarmOutput;
			
	//Rapportera upptagen enhet	
		oaksgvl.aBModbusBusyFlagga[modbusTCP.iModbusLoop,nUnitID] := bBusy;
		
ELSE
	bFAULT := TRUE;
END_IF

END_FUNCTION_BLOCK

// oaksModbusLibrary/Fidelix/FXIO (IO-kort)/Modulblock/fbFxIO_DO8
//Fidelix DO-16 IO-modul över ModbusTCP (används med t ex Moxa)
//Modulversion 1.10 / 2.20, funkar förhoppningsvis med senare versioner också
//Skrivning av DO, samt skrivning av fallback-konfiguration för DO. Om fallback för DO är till (nDOxfallback > 0) aktiveras det i modulen då ingen kommunikation skett efter 30 sekunder
//Robert H, Oaks. 23-09-13
//Ver. 1.1
//OBS se manual för FXIO: https://oaksab.sharepoint.com/sites/Utveckling/_layouts/15/Doc.aspx?sourcedoc={22bc18e8-aa49-48c1-a1e6-a272a7cd26b5}&action=edit&wd=target%28Integrationer.one%7C5ac70296-2750-4373-ab29-5663253fae71%2FFxIO%20%28Fidelix%20IO-kort%5C%29%7C584643fa-d9bd-4007-939c-93e7e7825215%2F%29&wdorigin=703
{attribute 'initialize_on_call'}
FUNCTION_BLOCK fbFxIO_DO8
VAR_INPUT
	bEnable 	: BOOL := TRUE; //Aktivering
	modbusTCP 	: ST_ModbusTCP;	//Modbus-konfiguration
	nUnitID		: BYTE := 0;	//Moduladress
	tTimeOut 	: TIME := T#5S;	//Kom. timeout
	bSetConfig	: BOOL := FALSE;//Skriv fallback-inställningar till modul
	
	{attribute 'initialize_on_call'}
	rbDO1 : REFERENCE TO BOOL;		//Digitalutgång 1
	nDO1fallback : BYTE := 0; 		//Fallback (0=Ej fallback, 1=Fallback 0, 2=Fallback 1);
	{attribute 'initialize_on_call'}
	rbDO2 : REFERENCE TO BOOL; 		//Digitalutgång 2
	nDO2fallback : BYTE := 0; 		//Fallback (0=Ej fallback, 1=Fallback 0, 2=Fallback 1);
	{attribute 'initialize_on_call'}
	rbDO3 : REFERENCE TO BOOL; 		//Digitalutgång 3
	nDO3fallback : BYTE := 0; 		//Fallback (0=Ej fallback, 1=Fallback 0, 2=Fallback 1);
	{attribute 'initialize_on_call'}
	rbDO4 : REFERENCE TO BOOL; 		//Digitalutgång 4
	nDO4fallback : BYTE := 0; 		//Fallback (0=Ej fallback, 1=Fallback 0, 2=Fallback 1);
	{attribute 'initialize_on_call'}
	rbDO5 : REFERENCE TO BOOL;		//Digitalutgång 5
	nDO5fallback : BYTE := 0; 		//Fallback (0=Ej fallback, 1=Fallback 0, 2=Fallback 1);
	{attribute 'initialize_on_call'}
	rbDO6 : REFERENCE TO BOOL;		//Digitalutgång 6
	nDO6fallback : BYTE := 0; 		//Fallback (0=Ej fallback, 1=Fallback 0, 2=Fallback 1);
	{attribute 'initialize_on_call'}
	rbDO7 : REFERENCE TO BOOL; 		//Digitalutgång 7
	nDO7fallback : BYTE := 0; 		//Fallback (0=Ej fallback, 1=Fallback 0, 2=Fallback 1);
	{attribute 'initialize_on_call'}
	rbDO8 : REFERENCE TO BOOL; 		//Digitalutgång 8
	nDO8fallback : BYTE := 0; 		//Fallback (0=Ej fallback, 1=Fallback 0, 2=Fallback 1);
END_VAR

VAR_OUTPUT
	sPV8 	: STRING;	//Modbus konfiguering
	bFAULT 	: BOOL;		//Kommunikationsfel
END_VAR
VAR
	sIP: STRING(255);
	sPort: STRING(255);
	sModbusID: STRING(255);
	sModbusLoop: STRING(255);
	sTemp : STRING(255);	

	bSekvensFlagga : BOOL;
	iStep: INT;
	bError: BOOL;
	bBusy: BOOL;

	fbKommTof : tof; 
	fbKommTon : fbAlarm;
	
	//Configuration
	FB_MBWriteRegs_Config: FB_MBWriteSingleReg;
	wWriteConfig : WORD; //Läs/skriv input regs modbus function 4.
		
	//Outputs
	FB_MBWriteRegs_Outputs: FB_MBWriteSingleReg;
	wWriteOutputs : WORD; //Läs/skriv input regs modbus function 6.
		
	R_TRIG_Sekvens: R_TRIG;
END_VAR

IF nUnitID <> 0 THEN
	//Sekvens
		R_TRIG_Sekvens(CLK:= oaksGVL.aBModbusSekvens[modbusTCP.iModbusLoop] = BYTE_TO_INT(nUnitID), Q=> bSekvensFlagga);
		
	//Modbus config
		sIP := CONCAT (modbusTCP.sIPAddr, '');
		sPort := CONCAT ('<br>Port: ', UINT_TO_STRING(modbusTCP.nTCPPort)); 								
		sModbusID := CONCAT('<br>ID: ', BYTE_TO_STRING(nUnitID));
		sModbusLoop := CONCAT('<br>Loop: ', INT_TO_STRING(modbusTCP.iModbusLoop));	
	
		sTemp := sIP;
		sTemp := CONCAT(sTemp, sPort);
		sTemp := CONCAT(sTemp, sModbusID);
		sTemp := CONCAT(sTemp, sModbusLoop);
		
		sPV8 := sTemp;
	
	//Läs- och skrivningar
		CASE iStep OF
	
		0: 	//Start/reset
			bBusy := FALSE;
							
			IF bEnable AND bSekvensFlagga THEN
				iStep := 1;
				bError := FALSE;
			END_IF
		
		1:	//Skriv fallback-inställningar vid bSetConfig
		wWriteConfig.0 := 	nDO1fallback = 2;	//LSB bit 0 är fallbackvärde för utgång 1
		wWriteConfig.8 := 	nDO1fallback > 0;	//MSB bit 0 är om fallback ska användas för utgång 1
		
		wWriteConfig.1 := 	nDO2fallback = 2;	//LSB bit 1 är fallbackvärde för utgång 2
		wWriteConfig.9 := 	nDO2fallback > 0;	//MSB bit 1 är om fallback ska användas för utgång 2
		
		wWriteConfig.2 := 	nDO3fallback = 2;	//Osv...
		wWriteConfig.10 := 	nDO3fallback > 0;
		
		wWriteConfig.3 := 	nDO4fallback = 2;
		wWriteConfig.11 := 	nDO4fallback > 0;
		
		wWriteConfig.4 := 	nDO5fallback = 2;
		wWriteConfig.12 := 	nDO5fallback > 0;
		
		wWriteConfig.5 := 	nDO6fallback = 2;
		wWriteConfig.13 := 	nDO6fallback > 0;
		
		wWriteConfig.6 := 	nDO7fallback = 2;
		wWriteConfig.14 := 	nDO7fallback > 0;
		
		wWriteConfig.7 := 	nDO8fallback = 2;
		wWriteConfig.15 := 	nDO8fallback > 0;	
		
		FB_MBWriteRegs_Config.bExecute := bSetConfig;
		
		FB_MBWriteRegs_Config(
			sIPAddr:= modbusTCP.sIpAddr, 
			nTCPPort:= modbusTCP.nTCPPort, 
			nUnitID:= nUnitID,
			nMBAddr:= 1,
			nValue:= wWriteConfig, 
			bExecute:= , 
			tTimeout:= tTimeout , 
			bBusy=> , 
			bError=> , 
			nErrId=> );
				
			IF FB_MBWriteRegs_Config.bError THEN
				FB_MBWriteRegs_Config(bExecute := FALSE);
				iStep := 99;
			END_IF
		
			//Next step
			IF NOT FB_MBWriteRegs_Config.bBusy AND NOT FB_MBWriteRegs_Config.bError THEN
				FB_MBWriteRegs_Config(bExecute := FALSE);
				bError := FALSE;
				iStep := 2;
			END_IF;
	
		2: //Skriv digitalutgångar från PLC
			bBusy := TRUE;	
				
			IF __ISVALIDREF(rbDO1) THEN wWriteOutputs.0 := rbDO1; END_IF
			IF __ISVALIDREF(rbDO2) THEN wWriteOutputs.1 := rbDO2; END_IF
			IF __ISVALIDREF(rbDO3) THEN wWriteOutputs.2 := rbDO3; END_IF
			IF __ISVALIDREF(rbDO4) THEN wWriteOutputs.3 := rbDO4; END_IF
			IF __ISVALIDREF(rbDO5) THEN wWriteOutputs.4 := rbDO5; END_IF
			IF __ISVALIDREF(rbDO6) THEN wWriteOutputs.5 := rbDO6; END_IF
			IF __ISVALIDREF(rbDO7) THEN wWriteOutputs.6 := rbDO7; END_IF
			IF __ISVALIDREF(rbDO8) THEN wWriteOutputs.7 := rbDO8; END_IF
			
			
			FB_MBWriteRegs_Outputs.bExecute := TRUE;
			
			FB_MBWriteRegs_Outputs(
				sIPAddr:= modbusTCP.sIpAddr, 
				nTCPPort:= modbusTCP.nTCPPort, 
				nUnitID:= nUnitID,
				nMBAddr:= 0,
				nValue:= wWriteOutputs, 
				bExecute:= , 
				tTimeout:= tTimeout , 
				bBusy=> , 
				bError=> , 
				nErrId=> );
					
			IF FB_MBWriteRegs_Outputs.bError THEN
				FB_MBWriteRegs_Outputs(bExecute := FALSE);
				iStep := 99;
			END_IF
		
			//Next step
			IF NOT FB_MBWriteRegs_Outputs.bBusy AND NOT FB_MBWriteRegs_Outputs.bError THEN
				FB_MBWriteRegs_Outputs(bExecute := FALSE);
				bError := FALSE;
				iStep := 20;
			END_IF;
	
		20: //Done
			bBusy := FALSE;
			iStep := 0;
			bSetConfig := FALSE;
	
		99: //Error handling
			bBusy := FALSE;
			bError := TRUE;
			iStep := 0;
			
	END_CASE
	
	//Kommunikationsfel modul
		fbKommTof(IN:=bError , PT:=T#20S , Q=> , ET=> );
		fbKommTon(bInput:=fbKommTof.Q , tAlarmDelay:=T#1M , bAutoReset:= , bAlarmOutput=> );
		bFAULT :=fbKommTon.bAlarmOutput;
			
	//Rapportera upptagen enhet	
		oaksgvl.aBModbusBusyFlagga[modbusTCP.iModbusLoop,nUnitID] := bBusy;
ELSE
	bFAULT := TRUE;
END_IF

END_FUNCTION_BLOCK

// oaksModbusLibrary/Fläktwoods/Spjällställdon/fbFlaktwoods227PMMB
//OAKS AB
//2020-03-17
//Funktionsblock för modbus-TCP, Fläktwoods 227PM-MB (Tryck). Fungerar även för fbGruner227PMxxMB.
FUNCTION_BLOCK fbFlaktwoods227PMMB
VAR_INPUT
	sIPAddr : STRING := ''; 
	nTCPPort : UINT;
	nUnitID : UINT :=1;
	iModbusLoop : INT :=1; //Modbusslinga	
	rSetpoint : REAL; //Börvärde
	iMode : INT; //Överstyrning spjälläge 0: None 1: Open 2: Close 3: Min 4: Max 5: Mid
	SP1 AT %M* : REAL;//Min-tryck~wp:[unit]Pa[format]0[trendoptions]i:300
	SP2 AT %M* : REAL;//Max-tryck~wp:[unit]Pa[format]0[trendoptions]i:300	
		
END_VAR
VAR_OUTPUT
	
	PV1 AT %M* : REAL;//Tryck~wp:[unit]Pa[format]0[trendoptions]i:300
	PV5 AT %M* : UINT;//Spjäll-läge 0: None 1: Open 2: Close 3: Min 4: Max 5: Mid~wp:[format]0[trendoptions]i:14400, t:1
	PV6 AT %M* : REAL;//Inställt min-tryck~wp:[unit]Pa[format]0[trendoptions]i:14400, t:1
	PV7 AT %M* : REAL;//Inställt max-tryck~wp:[unit]Pa[format]0[trendoptions]i:14400, t:1
	PV10 AT %M* : STRING;//Modbus konfiguering~wp:
	OP AT %M* : REAL;//Relativ position~wp:[unit]%[format]0[trendoptions]i:300
	CSP AT %M* : REAL;//Uträknat börvärde~wp:[unit]Pa[format]0[trendoptions]i:300
	FAULT AT %M* : BOOL;//Kommunikationsfel~wp:
	

END_VAR
VAR
	offset : WORD;
	rTemp : REAL;
	iTemp : UINT;
	wTemp : WORD;
	bSekvensFlagga : BOOL;
	
	FB_MBReadRegs_ArrHolding1: FB_MBReadRegs;
	ArrHolding1 : ARRAY [0..9] OF WORD; //Holding
	wActSetpoint : WORD; //Börvärde 0
	wModeOut : WORD; //Överstyrning 1 
	wRelPos : WORD; //Relativ position 5
	wAbsPress : WORD; //Volym 7

	FB_MBReadRegs_ArrHolding2 : FB_MBReadRegs;
	ArrHolding2 : ARRAY [99..122] OF WORD; //Holding	
	wAlarm : WORD; //Fel 105
	wMinPress : WORD; //Min setpoint 121
	wMaxPress : WORD; //Max setpoint 122
	
	FB_MBReadRegs_ArrHolding3 : FB_MBReadRegs;
	ArrHolding3 : ARRAY [120..122] OF WORD; //Holding	
		
	FB_MBWriteSingleReg_Setpoint : FB_MBWriteSingleReg; 
	FB_MBWriteSingleReg_Mode : FB_MBWriteSingleReg; 
	
	//Skrivning
	fbWriteHoldingDoubleControlledMin: fbDoubleControlledModbusHolding;
	fbWriteHoldingDoubleControlledMax: fbDoubleControlledModbusHolding;
	
	//Kommunikationsfel
	fbKommTof : tof; 
	fbKommTon : ton;
	
	fb_CSP : Tc3_BA.FB_BA_Chrct02;	
	
	sIP: STRING(255);
	sPort: STRING(255);
	sModbusID: STRING(255);
	sModbusLoop: STRING(255);
	
	sTemp: STRING(255);
END_VAR

//General
	offset := 0;
//Sekvens	
	bSekvensFlagga := oaksGVL.aBModbusSekvens[iModbusLoop] = UINT_TO_INT(nUnitID);
//Modbus konfiguering
	sIP := CONCAT (SIPAddr, '');
	sPort := CONCAT ('<br>Port: ', UINT_TO_STRING(nTCPPort)); 								
	sModbusID := CONCAT('<br>ID: ', UINT_TO_STRING(nUnitID));
	sModbusLoop := CONCAT('<br>Loop: ', INT_TO_STRING(iModbusLoop));

	sTemp := sIP;
	sTemp := CONCAT(sTemp, sPort);
	sTemp := CONCAT(sTemp, sModbusID);
	sTemp := CONCAT(sTemp, sModbusLoop);
		
	PV10 := sTemp;

///////////////		
//READ
///////////////		
	
	//Read Holding 0-8
	FB_MBReadRegs_ArrHolding1(
	sIPAddr:= sIpAddr, 
	nTCPPort:= INT_TO_UINT(nTCPPort), 
	nUnitID:= INT_TO_BYTE(nUnitID), 
	nQuantity:= 9, 
	nMBAddr:= 0 + offset, 
	cbLength:= SIZEOF(ArrHolding1), 
	pDestAddr:= ADR(ArrHolding1), 
	bExecute:= bSekvensFlagga, 
	tTimeout:= T#3S, 
	bBusy=> , 
	bError=> , 
	nErrId=> , 
	cbRead=> );
	
		//Values
		wActSetpoint := ArrHolding1[0]; //0
		wModeOut := ArrHolding1[1]; //1
		//ArrHolding1[2]; //2
		//ArrHolding1[3]; //3
		//ArrHolding1[4]; //4
		wRelPos := ArrHolding1[5]; //5
		//ArrHolding1[6]; //6
		wAbsPress := ArrHolding1[7]; //7
		//ArrHolding1[8]; //8
								
		//Absolute Volume flow
		//Converter from m2 to l/s
		iTemp := WORD_TO_UINT(wAbsPress);
		rTemp := UINT_TO_REAL(iTemp);
		PV1 := rTemp;
	
		//Relative Position
		iTemp := WORD_TO_UINT(wRelPos);
		rTemp := UINT_TO_REAL(iTemp);
		OP := rTemp / 100;
		
		//Actual damper-mode
		PV5 := wModeOut;
						
	//Read Holding 100-108
	FB_MBReadRegs_ArrHolding2(
	sIPAddr:= sIpAddr, 
	nTCPPort:= INT_TO_UINT(nTCPPort), 
	nUnitID:= INT_TO_BYTE(nUnitID), 
	nQuantity:= 9, 
	nMBAddr:= 100 + offset, 
	cbLength:= SIZEOF(ArrHolding2), 
	pDestAddr:= ADR(ArrHolding2), 
	bExecute:= bSekvensFlagga, 
	tTimeout:= T#3S, 
	bBusy=> , 
	bError=> , 
	nErrId=> , 
	cbRead=> );
	
		//Tilldela värden
		//ArrHolding2[100]; //100
		//ArrHolding2[101]; //101
		//ArrHolding2[102]; //102
		//ArrHolding2[103]; //103
		//ArrHolding2[104]; //104
		wAlarm := ArrHolding2[105]; //105
		//ArrHolding2[106]; //106
		//ArrHolding2[107]; //107
		//ArrHolding2[108]; //108

	//Read Holding 120-122
	FB_MBReadRegs_ArrHolding3(
	sIPAddr:= sIpAddr, 
	nTCPPort:= INT_TO_UINT(nTCPPort), 
	nUnitID:= INT_TO_BYTE(nUnitID), 
	nQuantity:= 3, 
	nMBAddr:= 120 + offset, 
	cbLength:= SIZEOF(ArrHolding3), 
	pDestAddr:= ADR(ArrHolding3), 
	bExecute:= bSekvensFlagga, 
	tTimeout:= T#3S, 
	bBusy=> , 
	bError=> , 
	nErrId=> , 
	cbRead=> );	
		
		
		wMinPress := ArrHolding3[120]; //120
		wMaxPress := ArrHolding3[121]; //121
		//ArrHolding3[122]; //122	
					
		//Setpoint pressure
		iTemp := WORD_TO_UINT(wMinPress);
		PV6 :=  UINT_TO_REAL(iTemp);
				
		//Setpoint pressure
		iTemp := WORD_TO_UINT(wMaxPress);
		PV7 := UINT_TO_REAL(iTemp);
		
	//Calculated setpoint
		fb_CSP(
			rX:= WORD_TO_REAL(wActSetpoint) / 100, 
			rX01:= 0, 
			rX02:= 100, 
			rY01:= PV6, 
			rY02:= PV7, 
			bLmt:= TRUE, 
			rY=> CSP, 
			bErr=> , 
			sErrDescr=> );
		
///////////////		
//WRITE
///////////////	
				
//Setpoint
	rTemp := LIMIT (0, rSetpoint, 100);
	wTemp := frealtoword(rTemp, 100);
	
	IF wTemp <> wActSetpoint AND bSekvensFlagga THEN
		FB_MBWriteSingleReg_Setpoint.bExecute := TRUE;
	ELSE
		FB_MBWriteSingleReg_Setpoint.bExecute := FALSE;
	END_IF
	
	//Write Setpoint
	FB_MBWriteSingleReg_Setpoint(
	sIPAddr:= sIpAddr, 
	nTCPPort:= INT_TO_UINT(nTCPPort), 
	nUnitID:= INT_TO_BYTE(nUnitID), 
	nMBAddr:= 0 + offset, 
	nValue:= wTemp, 
	bExecute:= , 
	tTimeout:= T#3S, 
	bBusy=> , 
	bError=> , 
	nErrId=> );
	
//Override

	iTemp := INT_TO_WORD(iMode);
	
	IF wModeOut <> iTemp AND bSekvensFlagga THEN 
		FB_MBWriteSingleReg_Mode.bExecute := TRUE;
	ELSE 
		FB_MBWriteSingleReg_Mode.bExecute := FALSE;
	END_IF
	
	//Write Mode
	FB_MBWriteSingleReg_Mode(
	sIPAddr:= sIpAddr, 
	nTCPPort:= INT_TO_UINT(nTCPPort), 
	nUnitID:= INT_TO_BYTE(nUnitID), 
	nMBAddr:= 1 + offset, 
	nValue:= UINT_TO_WORD(iTemp), 
	bExecute:= , 
	tTimeout:= T#3S, 
	bBusy=> , 
	bError=> , 
	nErrId=> );

//Read/write

//Min		
	fbWriteHoldingDoubleControlledMin(
	sIPAddr:= sIPAddr, 
	nTCPPort:= nTCPPort, 
	nUnitID:= UINT_TO_BYTE(nUnitID) , 
	nMBAddr:= 120+offset, 
	bExecute:=bSekvensFlagga , 
	rScale:= 1, 
	rWrite:= SP1, 
	bBusy=> , 
	bError=> );
//Max

			
	fbWriteHoldingDoubleControlledMax(
	sIPAddr:= sIPAddr, 
	nTCPPort:= nTCPPort, 
	nUnitID:= UINT_TO_BYTE(nUnitID) , 
	nMBAddr:= 121+offset, 
	bExecute:=bSekvensFlagga , 
	rScale:= 1, 
	rWrite:= SP2, 
	bBusy=> , 
	bError=> );
	

	
//Communication error
	fbKommTof(IN:=FB_MBReadRegs_ArrHolding1.bError , PT:=T#20S , Q=> , ET=> );
	fbKommTon(IN:=fbKommTof.Q , PT:=T#20M , Q=> , ET=> );
	FAULT :=fbKommTon.Q;
		
//Write busy	
	oaksgvl.aBModbusBusyFlagga[iModbusLoop,nUnitID] := FB_MBReadRegs_Arrholding1.bBusy OR FB_MBReadRegs_Arrholding2.bBusy OR FB_MBReadRegs_ArrHolding3.bBusy OR FB_MBWriteSingleReg_Setpoint.bBusy OR FB_MBWriteSingleReg_Mode.bBusy;

END_FUNCTION_BLOCK

// oaksModbusLibrary/Fläktwoods/Spjällställdon/fbFlaktwoods227VMMB
//OAKS AB
//2020-03-17
//Funktionsblock för modbus-TCP, Fläktwoods 227VM-MB (Flöde). Fungerar även för fbGruner227VMxxMB.
FUNCTION_BLOCK fbFlaktwoods227VMMB
VAR_INPUT
	sIPAddr : STRING := ''; 
	nTCPPort : UINT;
	nUnitID : UINT :=1;
	iModbusLoop : INT :=1; //Modbusslinga
	rSetpoint : REAL; //Börvärde
	iMode : INT; //Överstyrning spjälläge 0: None 1: Open 2: Close 3: Min 4: Max 5: Mid
	SP1 AT %M* : REAL;//Min-flöde~wp:[unit]l/s[format]0[trendoptions]i:300
	SP2 AT %M* : REAL;//Max-flöde~wp:[unit]l/s[format]0[trendoptions]i:300	
		
END_VAR
VAR_OUTPUT
	
	PV1 AT %M* : REAL;//Flöde~wp:[unit]l/s[format]0[trendoptions]i:300
	PV5 AT %M* : UINT;//Spjäll-läge 0: None 1: Open 2: Close 3: Min 4: Max 5: Mid~wp:[format]0[trendoptions]i:14400, t:1
	PV6 AT %M* : REAL;//Inställt min-flöde~wp:[unit]l/s[format]0[trendoptions]i:14400, t:1
	PV7 AT %M* : REAL;//Inställt max-flöde~wp:[unit]l/s[format]0[trendoptions]i:14400, t:1
	PV10 AT %M* : STRING;//Modbus konfiguering~wp:
	OP AT %M* : REAL;//Relativ position~wp:[unit]%[format]0[trendoptions]i:300
	CSP AT %M* : REAL;//Uträknat börvärde~wp:[unit]l/s[format]0[trendoptions]i:300
	FAULT AT %M* : BOOL;//Kommunikationsfel~wp:

END_VAR
VAR
	offset : WORD;
	rTemp : REAL;
	iTemp : UINT;
	wTemp : WORD;
	bSekvensFlagga : BOOL;
		
	FB_MBReadRegs_ArrHolding1: FB_MBReadRegs;
	ArrHolding1 : ARRAY [0..8] OF WORD; //Holding
	wActSetpoint : WORD; //Börvärde 0
	wModeOut : WORD; //Överstyrning 1 
	wRelPos : WORD; //Relativ position 5
	wAbsVolume : WORD; //Volym 7

	FB_MBReadRegs_ArrHolding2 : FB_MBReadRegs;
	ArrHolding2 : ARRAY [100..108] OF WORD; //Holding	
	wAlarm : WORD; //Fel 105
	wMinVolume : WORD; //Min setpoint 121
	wMaxVolume : WORD; //Max setpoint 122
	
	FB_MBReadRegs_ArrHolding3 : FB_MBReadRegs;
	ArrHolding3 : ARRAY [120..122] OF WORD; //Holding	
		
	FB_MBWriteSingleReg_Setpoint : FB_MBWriteSingleReg; 
	FB_MBWriteSingleReg_Mode : FB_MBWriteSingleReg; 
	
	//Skrivning
	fbWriteHoldingDoubleControlledMin: fbDoubleControlledModbusHolding;
	fbWriteHoldingDoubleControlledMax: fbDoubleControlledModbusHolding;

	
